	fbCoeRead(bExecute:= FALSE);
		IF NOT fbCoeRead.bBusy THEN					(* Baustein ist durchgelaufen *)
		IF fbCoeRead.bError THEN				(* Wenn ein Error vorliegt, wird dieser ausgegeben *)
			nLastErrIDTemp 
				:= fbCoeRead.nErrID;
			bCoeReadError := TRUE;
		ELSE
			IF nReadBuf.0 THEN
				arrSafetyKlemmeInfo[nAktKlemme].arrFehler[nFehlerIdx] := TRUE;
				arrSafetyKlemmeInfo[nAktKlemme].arrFehlertext[nFehlerIdx] := 
					CONCAT('Temperaturfehler der Safety-Klemme! Uebertemperatur µC1! Adresse: ',
						arrSafetyKlemmeInfo[nAktKlemme].sName);
				nFehlerIdx := nFehlerIdx + 1;
			END_IF	
			IF nReadBuf.1 THEN
				arrSafetyKlemmeInfo[nAktKlemme].arrFehler[nFehlerIdx] := TRUE;
				arrSafetyKlemmeInfo[nAktKlemme].arrFehlertext[nFehlerIdx] := 
					CONCAT('Temperaturfehler der Safety-Klemme! Uebertemperatur µC2! Adresse: ',
						arrSafetyKlemmeInfo[nAktKlemme].sName);
				nFehlerIdx := nFehlerIdx + 1;	
			END_IF	
			IF  nReadBuf.2 THEN
				arrSafetyKlemmeInfo[nAktKlemme].arrFehler[nFehlerIdx] := TRUE;
				arrSafetyKlemmeInfo[nAktKlemme].arrFehlertext[nFehlerIdx] := 
					CONCAT('Temperaturfehler der Safety-Klemme! Uebertemperatur der Ausgangsplatine! Adresse: ',
						arrSafetyKlemmeInfo[nAktKlemme].sName);
				nFehlerIdx := nFehlerIdx + 1;	
			END_IF	
			IF nReadBuf.3 THEN
				arrSafetyKlemmeInfo[nAktKlemme].arrFehler[nFehlerIdx] := TRUE;
				arrSafetyKlemmeInfo[nAktKlemme].arrFehlertext[nFehlerIdx] := 
					CONCAT('Temperaturfehler der Safety-Klemme! Untertemperatur µC1! Adresse: ',
						arrSafetyKlemmeInfo[nAktKlemme].sName);
				nFehlerIdx := nFehlerIdx + 1;	
			END_IF
			(*Fehler am Ausgang - Open Load oder Mindeststrom unterschritten / Höchststrom überschritten*)
			IF nReadBuf.4 THEN
				arrSafetyKlemmeInfo[nAktKlemme].arrFehler[nFehlerIdx] := TRUE;
				arrSafetyKlemmeInfo[nAktKlemme].arrFehlertext[nFehlerIdx] := 
					CONCAT('Temperaturfehler der Safety-Klemme! Untertemperatur µC1! Adresse: ',
						arrSafetyKlemmeInfo[nAktKlemme].sName);
				nFehlerIdx := nFehlerIdx + 1;	
			END_IF
			IF nReadBuf.5 THEN
				arrSafetyKlemmeInfo[nAktKlemme].arrFehler[nFehlerIdx] := TRUE;
				arrSafetyKlemmeInfo[nAktKlemme].arrFehlertext[nFehlerIdx] := 
					CONCAT('Temperaturfehler der Safety-Klemme! Untertemperatur der Ausgangsplatine! Adresse: ',
						arrSafetyKlemmeInfo[nAktKlemme].sName);
				nFehlerIdx := nFehlerIdx + 1;	
			END_IF	
			IF nReadBuf.6 THEN
				arrSafetyKlemmeInfo[nAktKlemme].arrFehler[nFehlerIdx] := TRUE;
				arrSafetyKlemmeInfo[nAktKlemme].arrFehlertext[nFehlerIdx] := 
					CONCAT('Temperaturfehler der Safety-Klemme! Temperaturdifferenz auf der Prozessorplatine ist zu groß! Adresse: ',
						arrSafetyKlemmeInfo[nAktKlemme].sName);
				nFehlerIdx := nFehlerIdx + 1;	
			END_IF	
			IF nReadBuf.7 THEN
				arrSafetyKlemmeInfo[nAktKlemme].arrFehler[nFehlerIdx] := TRUE;
				arrSafetyKlemmeInfo[nAktKlemme].arrFehlertext[nFehlerIdx] := 
					CONCAT('Temperaturfehler der Safety-Klemme! Temperaturdifferenz zwischen den Platinen ist zu groß! Adresse: ',
						arrSafetyKlemmeInfo[nAktKlemme].sName);
				nFehlerIdx := nFehlerIdx + 1;	
			END_IF	
			bCoeReadError := FALSE;
		END_IF
		nStateDatenAuslesen := 0;	
		arrSafetyKlemmeInfo[nAktKlemme].nAnzFehler := nFehlerIdx;
		nFehlerIdx := 0;
		bBusy := FALSE;	
	END_IF
END_CASE

sKlarTextCoeMeldung	:= F_AdsErrorIdToString(I_nErrorID:=nLastErrIDTemp);
END_ACTION

ACTION e_EL2911:

// 16#10F3 ist der Index für den Diag-History-Reiter in der online-Ansicht im EA-Baum
// 16#01: Subindex für das Maximum an Meldungen
// 16#02: Subindex für die neuste Meldung
// 16#03: Subindex für die neuste quittierte Meldung
// 16#04: Subindex eine neue Meldung vorhanden
// 16#05: Subindex für allgemeine Flags
// 16#06 - 16#45: Subindexe für die Meldungen

// Weitere Diagnoseobjekte:
// 16#F984 ist der Index für Device System Data vom Controller 1
// 16#02: Subindex für die Temperatur
// 16#F985 ist der Index für Device System Data vom Controller 2
// 16#02: Subindex für die Temperatur
// Sollten aber auch alle in der Diag History stehen.

// ModuleFault:
// 16#6002:01 Ch1
// 16#6012:01 Ch2
// 16#6022:01 Ch3
// 16#6032:01 Ch4
// 16#6042:01 Ch5
// 16#6052:01 Ch6
// 16#6062:01 Ch7
// 16#6072:01 Ch8

// Eine richtige Diagnose der TwinSAFE-Ein-/ und Ausgänge ist nicht mehr über die CoE-Objekte möglich. Das muss über die DiagHistory gemacht werden. GGf. ist das bald in der HMI
CASE nStateDatenAuslesen OF
	
0:	// EL2912 Diagnose init 
	bBusy 			:= TRUE;	// Solange diese Bit an ist, wird diese Aktion aufgerufen
	nChannelDiag	:= 1;	// Immer bei Kanal 1 beginnen.
	MEMSET(ADR(arrModuleFault),0,SIZEOF(arrModuleFault));	// Rücksetzen
	MEMSET(ADR(arrModuleFaultLink),0,SIZEOF(arrModuleFaultLink));	// Rücksetzen
	
	nStateDatenAuslesen	:= nStateDatenAuslesen +1;
	
1:	// Module Fault der einzelnen Kanäle auslesen: Index errechnen
	
	nCoeIndex		:= 16#6002 + ((nChannelDiag-1)* 16#10);	// Index für ModuleFault pro Kanal
	nCoESubIndex	:= 16#01;	// Index der neusten Meldung
	nStateDatenAuslesen	:= nStateDatenAuslesen +1;
	
2:	// Module Fault der einzelnen Kanäle auslesen: Lesen starten

	fbCoeRead(
		sNetId		:= sEtherCatNetID,
		nSlaveAddr 	:= arrSafetyKlemmeInfo[nAktKlemme].nAdresse,
		nIndex		:= nCoEIndex,
		nSubIndex 	:= nCoESubIndex,
		pDstBuf		:= ADR(nDiagMessage),
		cbBufLen		:= SIZEOF(nDiagMessage),
		bExecute		:= TRUE,

		bError		=> bCoeReadError,
		nErrId		=> nCoeReadErrId
	);
	nStateDatenAuslesen := nStateDatenAuslesen + 1;

3:	// Module Fault der einzelnen Kanäle auslesen: Warten auf gelesen

	fbCoeRead(bExecute:= FALSE);

	IF NOT fbCoeRead.bBusy
	THEN	// Baustein ist durchgelaufen
		IF fbCoeRead.bError
		THEN	// Wenn ein Error vorliegt, wird dieser ausgegeben
			nLastErrIDTemp := fbCoeRead.nErrID;	// Error-ID des CoE Reads wird gespeichert
			bCoeReadError := TRUE;
		ELSE
			bCoeReadError := FALSE;
		END_IF
		
		nStateDatenAuslesen := nStateDatenAuslesen + 1;
	END_IF
	
4:	// Module Fault der einzelnen Kanäle auslesen: Lesen auswerten

	arrModuleFault[nChannelDiag]	:= nDiagMessage <> 0;
	
	IF nChannelDiag = 1
	THEN
		nStateDatenAuslesen := 11;
		nChannelDiag	:= 1;
	ELSE
		nChannelDiag	:= nChannelDiag +1;
		nStateDatenAuslesen := 1;
	END_IF

11:	// Module Fault Link der einzelnen Kanäle auslesen: Index errechnen

// ModuleFaultLink:
// 16#8000:07 Ch1
// 16#8010:07 Ch2
// 16#8020:07 Ch3
// 16#8030:07 Ch4
// 16#8040:07 Ch5
// 16#8050:07 Ch6
// 16#8060:07 Ch7
// 16#8070:07 Ch8

	nCoeIndex		:= 16#8000 + ((nChannelDiag-1)* 16#10);	// Index für ModuleFaultLink pro Kanal
	nCoESubIndex	:= 16#07;
	nStateDatenAuslesen	:= nStateDatenAuslesen +1;
	
12:	// Module Fault Link der einzelnen Kanäle auslesen: Lesen starten

	fbCoeRead(
		sNetId		:= sEtherCatNetID,
		nSlaveAddr 	:= arrSafetyKlemmeInfo[nAktKlemme].nAdresse,
		nIndex		:= nCoEIndex,
		nSubIndex 	:= nCoESubIndex,
		pDstBuf		:= ADR(nDiagMessage),
		cbBufLen		:= SIZEOF(nDiagMessage),
		bExecute		:= TRUE,

		bError		=> bCoeReadError,
		nErrId		=> nCoeReadErrId
	);
	nStateDatenAuslesen := nStateDatenAuslesen + 1;

13:	// Module Fault Link der einzelnen Kanäle auslesen: Warten auf gelesen

	fbCoeRead(bExecute:= FALSE);

	IF NOT fbCoeRead.bBusy
	THEN	// Baustein ist durchgelaufen
		IF fbCoeRead.bError
		THEN	// Wenn ein Error vorliegt, wird dieser ausgegeben
			nLastErrIDTemp := fbCoeRead.nErrID;	// Error-ID des CoE Reads wird gespeichert
			bCoeReadError := TRUE;
		ELSE
			bCoeReadError := FALSE;
		END_IF
		
		nStateDatenAuslesen := nStateDatenAuslesen + 1;
	END_IF
	
14:	// Module Fault Link der einzelnen Kanäle auslesen: Lesen auswerten

	arrModuleFaultLink[nChannelDiag]	:= nDiagMessage <> 0;
	
	IF nChannelDiag = 1
	THEN
		nStateDatenAuslesen := 21;
		nChannelDiag	:= 1;
	ELSE
		nChannelDiag	:= nChannelDiag +1;
		nStateDatenAuslesen := 11;
	END_IF
	
21:	// ModuleFault gesammelt auswerten.

	bModuleFaultActive	:= FALSE;
	FOR nChannelDiag := 1 TO 1 DO
		IF arrModuleFault[nChannelDiag]
		THEN
			bModuleFaultActive	:= TRUE;
		END_IF
	END_FOR
	
	nStateDatenAuslesen := nStateDatenAuslesen + 1;
	
22:	// Fehlermeldung auswerten

	FOR nChannelDiag := 1 TO 1 DO
		IF arrModuleFault[nChannelDiag]
			AND arrModuleFaultLink[nChannelDiag]
		THEN	// Modulfehler mit aktivem ModuleFaultLink
		
			arrSafetyKlemmeInfo[nAktKlemme].arrFehler[nFehlerIdx] := TRUE;
			arrSafetyKlemmeInfo[nAktKlemme].arrFehlertext[nFehlerIdx] := 
				CONCAT('ModuleFault bei Klemme: ',
				CONCAT(arrSafetyKlemmeInfo[nAktKlemme].sName,
				CONCAT(' Kanal: ',
				CONCAT(TO_STRING(nChannelDiag),' Bei aktivem ModuleFaultLink. Der Fehler kann aber auch an einem anderen Kanal liegen.'))));
			nFehlerIdx := nFehlerIdx + 1;
		ELSIF arrModuleFault[nChannelDiag]
		THEN	// Modulfehler ohne ModuleFaultLink. Das heißt, dass der Fehler definitiv an diesem Kanal liegt.
		
			arrSafetyKlemmeInfo[nAktKlemme].arrFehler[nFehlerIdx] := TRUE;
			arrSafetyKlemmeInfo[nAktKlemme].arrFehlertext[nFehlerIdx] := 
				CONCAT('ModuleFault bei Klemme: ',
				CONCAT(arrSafetyKlemmeInfo[nAktKlemme].sName,
				CONCAT(' Kanal: ',TO_STRING(nChannelDiag))));
			nFehlerIdx := nFehlerIdx + 1;
		END_IF
	END_FOR
	
	nStateDatenAuslesen := 99;	// Fertig
	
99:	// Fertig mit auslesen
	
	arrSafetyKlemmeInfo[nAktKlemme].nAnzFehler := nFehlerIdx;
	nStateDatenAuslesen := 0;
	nFehlerIdx := 0; 
	bBusy := FALSE;

END_CASE
END_ACTION

ACTION e_EL2912:

// 16#10F3 ist der Index für den Diag-History-Reiter in der online-Ansicht im EA-Baum
// 16#01: Subindex für das Maximum an Meldungen
// 16#02: Subindex für die neuste Meldung
// 16#03: Subindex für die neuste quittierte Meldung
// 16#04: Subindex eine neue Meldung vorhanden
// 16#05: Subindex für allgemeine Flags
// 16#06 - 16#45: Subindexe für die Meldungen

// Weitere Diagnoseobjekte:
// 16#F984 ist der Index für Device System Data vom Controller 1
// 16#02: Subindex für die Temperatur
// 16#F985 ist der Index für Device System Data vom Controller 2
// 16#02: Subindex für die Temperatur
// Sollten aber auch alle in der Diag History stehen.

// ModuleFault:
// 16#6002:01 Ch1
// 16#6012:01 Ch2
// 16#6022:01 Ch3
// 16#6032:01 Ch4
// 16#6042:01 Ch5
// 16#6052:01 Ch6
// 16#6062:01 Ch7
// 16#6072:01 Ch8

// Eine richtige Diagnose der TwinSAFE-Ein-/ und Ausgänge ist nicht mehr über die CoE-Objekte möglich. Das muss über die DiagHistory gemacht werden. GGf. ist das bald in der HMI
CASE nStateDatenAuslesen OF
	
0:	// EL2912 Diagnose init 
	bBusy 			:= TRUE;	// Solange diese Bit an ist, wird diese Aktion aufgerufen
	nChannelDiag	:= 1;	// Immer bei Kanal 1 beginnen.
	MEMSET(ADR(arrModuleFault),0,SIZEOF(arrModuleFault));	// Rücksetzen
	MEMSET(ADR(arrModuleFaultLink),0,SIZEOF(arrModuleFaultLink));	// Rücksetzen
	
	nStateDatenAuslesen	:= nStateDatenAuslesen +1;
	
1:	// Module Fault der einzelnen Kanäle auslesen: Index errechnen
	
	nCoeIndex		:= 16#6002 + ((nChannelDiag-1)* 16#10);	// Index für ModuleFault pro Kanal
	nCoESubIndex	:= 16#01;	// Index der neusten Meldung
	nStateDatenAuslesen	:= nStateDatenAuslesen +1;
	
2:	// Module Fault der einzelnen Kanäle auslesen: Lesen starten

	fbCoeRead(
		sNetId		:= sEtherCatNetID,
		nSlaveAddr 	:= arrSafetyKlemmeInfo[nAktKlemme].nAdresse,
		nIndex		:= nCoEIndex,
		nSubIndex 	:= nCoESubIndex,
		pDstBuf		:= ADR(nDiagMessage),
		cbBufLen		:= SIZEOF(nDiagMessage),
		bExecute		:= TRUE,

		bError		=> bCoeReadError,
		nErrId		=> nCoeReadErrId
	);
	nStateDatenAuslesen := nStateDatenAuslesen + 1;

3:	// Module Fault der einzelnen Kanäle auslesen: Warten auf gelesen

	fbCoeRead(bExecute:= FALSE);

	IF NOT fbCoeRead.bBusy
	THEN	// Baustein ist durchgelaufen
		IF fbCoeRead.bError
		THEN	// Wenn ein Error vorliegt, wird dieser ausgegeben
			nLastErrIDTemp := fbCoeRead.nErrID;	// Error-ID des CoE Reads wird gespeichert
			bCoeReadError := TRUE;
		ELSE
			bCoeReadError := FALSE;
		END_IF
		
		nStateDatenAuslesen := nStateDatenAuslesen + 1;
	END_IF
	
4:	// Module Fault der einzelnen Kanäle auslesen: Lesen auswerten

	arrModuleFault[nChannelDiag]	:= nDiagMessage <> 0;
	
	IF nChannelDiag = 2
	THEN
		nStateDatenAuslesen := 11;
		nChannelDiag	:= 1;
	ELSE
		nChannelDiag	:= nChannelDiag +1;
		nStateDatenAuslesen := 1;
	END_IF

11:	// Module Fault Link der einzelnen Kanäle auslesen: Index errechnen

// ModuleFaultLink:
// 16#8000:07 Ch1
// 16#8010:07 Ch2
// 16#8020:07 Ch3
// 16#8030:07 Ch4
// 16#8040:07 Ch5
// 16#8050:07 Ch6
// 16#8060:07 Ch7
// 16#8070:07 Ch8

	nCoeIndex		:= 16#8000 + ((nChannelDiag-1)* 16#10);	// Index für ModuleFaultLink pro Kanal
	nCoESubIndex	:= 16#07;
	nStateDatenAuslesen	:= nStateDatenAuslesen +1;
	
12:	// Module Fault Link der einzelnen Kanäle auslesen: Lesen starten

	fbCoeRead(
		sNetId		:= sEtherCatNetID,
		nSlaveAddr 	:= arrSafetyKlemmeInfo[nAktKlemme].nAdresse,
		nIndex		:= nCoEIndex,
		nSubIndex 	:= nCoESubIndex,
		pDstBuf		:= ADR(nDiagMessage),
		cbBufLen		:= SIZEOF(nDiagMessage),
		bExecute		:= TRUE,

		bError		=> bCoeReadError,
		nErrId		=> nCoeReadErrId
	);
	nStateDatenAuslesen := nStateDatenAuslesen + 1;

13:	// Module Fault Link der einzelnen Kanäle auslesen: Warten auf gelesen

	fbCoeRead(bExecute:= FALSE);

	IF NOT fbCoeRead.bBusy
	THEN	// Baustein ist durchgelaufen
		IF fbCoeRead.bError
		THEN	// Wenn ein Error vorliegt, wird dieser ausgegeben
			nLastErrIDTemp := fbCoeRead.nErrID;	// Error-ID des CoE Reads wird gespeichert
			bCoeReadError := TRUE;
		ELSE
			bCoeReadError := FALSE;
		END_IF
		
		nStateDatenAuslesen := nStateDatenAuslesen + 1;
	END_IF
	
14:	// Module Fault Link der einzelnen Kanäle auslesen: Lesen auswerten

	arrModuleFaultLink[nChannelDiag]	:= nDiagMessage <> 0;
	
	IF nChannelDiag = 2
	THEN
		nStateDatenAuslesen := 21;
		nChannelDiag	:= 1;
	ELSE
		nChannelDiag	:= nChannelDiag +1;
		nStateDatenAuslesen := 11;
	END_IF
	
21:	// ModuleFault gesammelt auswerten.

	bModuleFaultActive	:= FALSE;
	FOR nChannelDiag := 1 TO 2 DO
		IF arrModuleFault[nChannelDiag]
		THEN
			bModuleFaultActive	:= TRUE;
		END_IF
	END_FOR
	
	nStateDatenAuslesen := nStateDatenAuslesen + 1;
	
22:	// Fehlermeldung auswerten

	FOR nChannelDiag := 1 TO 2 DO
		IF arrModuleFault[nChannelDiag]
			AND arrModuleFaultLink[nChannelDiag]
		THEN	// Modulfehler mit aktivem ModuleFaultLink
		
			arrSafetyKlemmeInfo[nAktKlemme].arrFehler[nFehlerIdx] := TRUE;
			arrSafetyKlemmeInfo[nAktKlemme].arrFehlertext[nFehlerIdx] := 
				CONCAT('ModuleFault bei Klemme: ',
				CONCAT(arrSafetyKlemmeInfo[nAktKlemme].sName,
				CONCAT(' Kanal: ',
				CONCAT(TO_STRING(nChannelDiag),' Bei aktivem ModuleFaultLink. Der Fehler kann aber auch an einem anderen Kanal liegen.'))));
			nFehlerIdx := nFehlerIdx + 1;
		ELSIF arrModuleFault[nChannelDiag]
		THEN	// Modulfehler ohne ModuleFaultLink. Das heißt, dass der Fehler definitiv an diesem Kanal liegt.
		
			arrSafetyKlemmeInfo[nAktKlemme].arrFehler[nFehlerIdx] := TRUE;
			arrSafetyKlemmeInfo[nAktKlemme].arrFehlertext[nFehlerIdx] := 
				CONCAT('ModuleFault bei Klemme: ',
				CONCAT(arrSafetyKlemmeInfo[nAktKlemme].sName,
				CONCAT(' Kanal: ',TO_STRING(nChannelDiag))));
			nFehlerIdx := nFehlerIdx + 1;
		END_IF
	END_FOR
	
	nStateDatenAuslesen := 99;	// Fertig
	
99:	// Fertig mit auslesen
	
	arrSafetyKlemmeInfo[nAktKlemme].nAnzFehler := nFehlerIdx;
	nStateDatenAuslesen := 0;
	nFehlerIdx := 0; 
	bBusy := FALSE;

END_CASE
END_ACTION

ACTION e_EP2918:

// 16#10F3 ist der Index für den Diag-History-Reiter in der online-Ansicht im EA-Baum
// 16#01: Subindex für das Maximum an Meldungen
// 16#02: Subindex für die neuste Meldung
// 16#03: Subindex für die neuste quittierte Meldung
// 16#04: Subindex eine neue Meldung vorhanden
// 16#05: Subindex für allgemeine Flags
// 16#06 - 16#45: Subindexe für die Meldungen

// Weitere Diagnoseobjekte:
// 16#F984 ist der Index für Device System Data vom Controller 1
// 16#02: Subindex für die Temperatur
// 16#F985 ist der Index für Device System Data vom Controller 2
// 16#02: Subindex für die Temperatur
// Sollten aber auch alle in der Diag History stehen.

// ModuleFault:
// 16#6002:01 Ch1
// 16#6012:01 Ch2
// 16#6022:01 Ch3
// 16#6032:01 Ch4
// 16#6042:01 Ch5
// 16#6052:01 Ch6
// 16#6062:01 Ch7
// 16#6072:01 Ch8

// Eine richtige Diagnose der TwinSAFE-Ein-/ und Ausgänge ist nicht mehr über die CoE-Objekte möglich. Das muss über die DiagHistory gemacht werden. GGf. ist das bald in der HMI
CASE nStateDatenAuslesen OF
	
0:	// EL2912 Diagnose init 
	bBusy 			:= TRUE;	// Solange diese Bit an ist, wird diese Aktion aufgerufen
	nChannelDiag	:= 1;	// Immer bei Kanal 1 beginnen.
	MEMSET(ADR(arrModuleFault),0,SIZEOF(arrModuleFault));	// Rücksetzen
	MEMSET(ADR(arrModuleFaultLink),0,SIZEOF(arrModuleFaultLink));	// Rücksetzen
	
	nStateDatenAuslesen	:= nStateDatenAuslesen +1;
	
1:	// Module Fault der einzelnen Kanäle auslesen: Index errechnen
	
	nCoeIndex		:= 16#6002 + ((nChannelDiag-1)* 16#10);	// Index für ModuleFault pro Kanal
	nCoESubIndex	:= 16#01;	// Index der neusten Meldung
	nStateDatenAuslesen	:= nStateDatenAuslesen +1;
	
2:	// Module Fault der einzelnen Kanäle auslesen: Lesen starten

	fbCoeRead(
		sNetId		:= sEtherCatNetID,
		nSlaveAddr 	:= arrSafetyKlemmeInfo[nAktKlemme].nAdresse,
		nIndex		:= nCoEIndex,
		nSubIndex 	:= nCoESubIndex,
		pDstBuf		:= ADR(nDiagMessage),
		cbBufLen		:= SIZEOF(nDiagMessage),
		bExecute		:= TRUE,

		bError		=> bCoeReadError,
		nErrId		=> nCoeReadErrId
	);
	nStateDatenAuslesen := nStateDatenAuslesen + 1;

3:	// Module Fault der einzelnen Kanäle auslesen: Warten auf gelesen

	fbCoeRead(bExecute:= FALSE);

	IF NOT fbCoeRead.bBusy
	THEN	// Baustein ist durchgelaufen
		IF fbCoeRead.bError
		THEN	// Wenn ein Error vorliegt, wird dieser ausgegeben
			nLastErrIDTemp := fbCoeRead.nErrID;	// Error-ID des CoE Reads wird gespeichert
			bCoeReadError := TRUE;
		ELSE
			bCoeReadError := FALSE;
		END_IF
		
		nStateDatenAuslesen := nStateDatenAuslesen + 1;
	END_IF
	
4:	// Module Fault der einzelnen Kanäle auslesen: Lesen auswerten

	arrModuleFault[nChannelDiag]	:= nDiagMessage <> 0;
	
	IF nChannelDiag = 8
	THEN
		nStateDatenAuslesen := 11;
		nChannelDiag	:= 1;
	ELSE
		nChannelDiag	:= nChannelDiag +1;
		nStateDatenAuslesen := 1;
	END_IF

11:	// Module Fault Link der einzelnen Kanäle auslesen: Index errechnen

// ModuleFaultLink:
// 16#8000:07 Ch1
// 16#8010:07 Ch2
// 16#8020:07 Ch3
// 16#8030:07 Ch4
// 16#8040:07 Ch5
// 16#8050:07 Ch6
// 16#8060:07 Ch7
// 16#8070:07 Ch8

	nCoeIndex		:= 16#8000 + ((nChannelDiag-1)* 16#10);	// Index für ModuleFaultLink pro Kanal
	nCoESubIndex	:= 16#07;
	nStateDatenAuslesen	:= nStateDatenAuslesen +1;
	
12:	// Module Fault Link der einzelnen Kanäle auslesen: Lesen starten

	fbCoeRead(
		sNetId		:= sEtherCatNetID,
		nSlaveAddr 	:= arrSafetyKlemmeInfo[nAktKlemme].nAdresse,
		nIndex		:= nCoEIndex,
		nSubIndex 	:= nCoESubIndex,
		pDstBuf		:= ADR(nDiagMessage),
		cbBufLen		:= SIZEOF(nDiagMessage),
		bExecute		:= TRUE,

		bError		=> bCoeReadError,
		nErrId		=> nCoeReadErrId
	);
	nStateDatenAuslesen := nStateDatenAuslesen + 1;

13:	// Module Fault Link der einzelnen Kanäle auslesen: Warten auf gelesen

	fbCoeRead(bExecute:= FALSE);

	IF NOT fbCoeRead.bBusy
	THEN	// Baustein ist durchgelaufen
		IF fbCoeRead.bError
		THEN	// Wenn ein Error vorliegt, wird dieser ausgegeben
			nLastErrIDTemp := fbCoeRead.nErrID;	// Error-ID des CoE Reads wird gespeichert
			bCoeReadError := TRUE;
		ELSE
			bCoeReadError := FALSE;
		END_IF
		
		nStateDatenAuslesen := nStateDatenAuslesen + 1;
	END_IF
	
14:	// Module Fault Link der einzelnen Kanäle auslesen: Lesen auswerten

	arrModuleFaultLink[nChannelDiag]	:= nDiagMessage <> 0;
	
	IF nChannelDiag = 8
	THEN
		nStateDatenAuslesen := 21;
		nChannelDiag	:= 1;
	ELSE
		nChannelDiag	:= nChannelDiag +1;
		nStateDatenAuslesen := 11;
	END_IF
	
21:	// ModuleFault gesammelt auswerten.

	bModuleFaultActive	:= FALSE;
	FOR nChannelDiag := 1 TO 8 DO
		IF arrModuleFault[nChannelDiag]
		THEN
			bModuleFaultActive	:= TRUE;
		END_IF
	END_FOR
	
	nStateDatenAuslesen := nStateDatenAuslesen + 1;
	
22:	// Fehlermeldung auswerten

	FOR nChannelDiag := 1 TO 8 DO
		IF arrModuleFault[nChannelDiag]
			AND arrModuleFaultLink[nChannelDiag]
		THEN	// Modulfehler mit aktivem ModuleFaultLink
		
			arrSafetyKlemmeInfo[nAktKlemme].arrFehler[nFehlerIdx] := TRUE;
			arrSafetyKlemmeInfo[nAktKlemme].arrFehlertext[nFehlerIdx] := 
				CONCAT('ModuleFault bei Klemme: ',
				CONCAT(arrSafetyKlemmeInfo[nAktKlemme].sName,
				CONCAT(' Kanal: ',
				CONCAT(TO_STRING(nChannelDiag),' Bei aktivem ModuleFaultLink. Der Fehler kann aber auch an einem anderen Kanal liegen.'))));
			nFehlerIdx := nFehlerIdx + 1;
		ELSIF arrModuleFault[nChannelDiag]
		THEN	// Modulfehler ohne ModuleFaultLink. Das heißt, dass der Fehler definitiv an diesem Kanal liegt.
		
			arrSafetyKlemmeInfo[nAktKlemme].arrFehler[nFehlerIdx] := TRUE;
			arrSafetyKlemmeInfo[nAktKlemme].arrFehlertext[nFehlerIdx] := 
				CONCAT('ModuleFault bei Klemme: ',
				CONCAT(arrSafetyKlemmeInfo[nAktKlemme].sName,
				CONCAT(' Kanal: ',TO_STRING(nChannelDiag))));
			nFehlerIdx := nFehlerIdx + 1;
		END_IF
	END_FOR
	
	nStateDatenAuslesen := 99;	// Fertig
	
99:	// Fertig mit auslesen
	
	arrSafetyKlemmeInfo[nAktKlemme].nAnzFehler := nFehlerIdx;
	nStateDatenAuslesen := 0;
	nFehlerIdx := 0; 
	bBusy := FALSE;

END_CASE
END_ACTION

ACTION f_AX5805:
CASE nStateDatenAuslesen OF
0:
	(*Auslesen der Anzahl der Achsen*)
	bBusy				:= TRUE;	
	nCoeIndex		:= 16#2F00; (*Anzahl der Achsen*)
	nCoESubIndex	:= 16#1;
	
	fbCoeRead(
	sNetId		:= sEtherCatNetID,
	nSlaveAddr 	:= arrSafetyKlemmeInfo[nAktKlemme].nAdresse,
	nIndex		:= nCoEIndex,
	nSubIndex 	:= nCoESubIndex,
	pDstBuf		:= ADR(nReadBuf),
	cbBufLen		:= SIZEOF(nReadBuf),
	bExecute		:= TRUE,

	bError		=> bCoeReadError,
	nErrId		=> nCoeReadErrId
	);
	
	fbCoeRead(bExecute:= FALSE);
	nAnzahlAchsen := UDINT_TO_INT(nReadBuf);
	
	IF NOT fbCoeRead.bBusy THEN
		nStateDatenAuslesen := nStateDatenAuslesen + 1;
	END_IF

1:	
	IF nAktAChse < nAnzahlAchsen THEN
		IF nAktAchse = 0 THEN
			  nAktAchse := 1;
	   END_IF
		
		nCoeIndex		:= 16#FA10; (*Grund der Abschaltung*)
		IF nAktAchse = 1 THEN 
			nCoESubIndex := 16#07;	(*Index Achse 1*)
		ELSE
			nCoeSubIndex := 16#08;	(*Index Achse 2*)
		END_IF
		 
		 fbCoeRead(
		 sNetId		:= sEtherCatNetID,
		 nSlaveAddr := arrSafetyKlemmeInfo[nAktKlemme].nAdresse,
		 nIndex		:= nCoEIndex,
		 nSubIndex 	:= nCoESubIndex,
		 pDstBuf		:= ADR(nReadBuf),
		 cbBufLen		:= SIZEOF(nReadBuf),
		 bExecute		:= TRUE,
	 
		 bError		=> bCoeReadError,
		 nErrId		=> nCoeReadErrId
		 );
			 
		 fbCoeRead(bExecute:= FALSE);
	 
		 IF NOT fbCoeRead.bBusy THEN				(* Baustein ist durchgelaufen *)
			 IF fbCoeRead.bError THEN				(* Wenn ein Error vorliegt, wird dieser ausgegeben; 0 = kein Fehler, 1= Eingang 1; 2= Eingang 2; 3= Eingang 3; 4 = Eingang 4*)
				 nLastErrIDTemp 
					 := fbCoeRead.nErrID;
				 bCoeReadError := TRUE;
			 ELSE
		 (*Fehler-Meldungen - Grund der Abschaltung CoE Objekt 0xFA10:07 und 0xFA10:08*)
		 (*Fehlermeldung aus AX5805.pdf Stand 03.12.2013 - S.101*)
			IF nReadBuf >= 16#100
			 AND nReadBuf < 16#200 THEN
				arrSafetyKlemmeInfo[nAktKlemme].arrFehler[nFehlerIdx] := TRUE;
				arrSafetyKlemmeInfo[nAktKlemme].arrFehlertext[nFehlerIdx] := 
					 CONCAT('AX5805: Das Statuswort wurde falsch berechnet! Achse: ',
					 CONCAT(INT_TO_STRING(nAktAchse),
					 CONCAT('Adresse: ',
						arrSafetyKlemmeInfo[nAktKlemme].sName)));
				nFehlerIdx := nFehlerIdx + 1;
			ELSIF nReadBuf >= 16#200
			 AND nReadBuf < 16#300 THEN
				arrSafetyKlemmeInfo[nAktKlemme].arrFehler[nFehlerIdx] := TRUE;
				arrSafetyKlemmeInfo[nAktKlemme].arrFehlertext[nFehlerIdx] := 
					 CONCAT('AX5805: Die Parameter sind fehlerhaft, wurden noch nicht geladen oder der AX5805 wurde noch nicht zurueckgesetzt (Error_Ack)! Achse: ',
					 CONCAT(INT_TO_STRING(nAktAchse),
					 CONCAT('Adresse: ',
						arrSafetyKlemmeInfo[nAktKlemme].sName)));
				nFehlerIdx := nFehlerIdx + 1;	
			ELSIF nReadBuf >= 16#300
			 AND nReadBuf < 16#400 THEN
				arrSafetyKlemmeInfo[nAktKlemme].arrFehler[nFehlerIdx] := TRUE;
				arrSafetyKlemmeInfo[nAktKlemme].arrFehlertext[nFehlerIdx] := 
					 CONCAT('AX5805: FSOE-Protokoll nicht im State DATA! Achse: ',
					 CONCAT(INT_TO_STRING(nAktAchse),
					 CONCAT('Adresse: ',
						arrSafetyKlemmeInfo[nAktKlemme].sName)));
				nFehlerIdx := nFehlerIdx + 1;
			ELSIF nReadBuf >= 16#400
			 AND nReadBuf < 16#500 THEN
				arrSafetyKlemmeInfo[nAktKlemme].arrFehler[nFehlerIdx] := TRUE;
				arrSafetyKlemmeInfo[nAktKlemme].arrFehlertext[nFehlerIdx] := 
					 CONCAT('AX5805: FSOE-Protokoll nicht im State DATA! Achse: ',
					 CONCAT(INT_TO_STRING(nAktAchse),
					 CONCAT('Adresse: ',
						arrSafetyKlemmeInfo[nAktKlemme].sName)));
				nFehlerIdx := nFehlerIdx + 1;
			 ELSIF nReadBuf >= 16#500
				 AND nReadBuf < 16#600 THEN
					 arrSafetyKlemmeInfo[nAktKlemme].arrFehler[nFehlerIdx] := TRUE;
					 arrSafetyKlemmeInfo[nAktKlemme].arrFehlertext[nFehlerIdx] := 
						  CONCAT('AX5805: FSOE-Protokoll nicht im State DATA! Achse: ',
						  CONCAT(INT_TO_STRING(nAktAchse),
						  CONCAT('Adresse: ',
							 arrSafetyKlemmeInfo[nAktKlemme].sName)));	
					 nFehlerIdx := nFehlerIdx + 1;
			 ELSIF nReadBuf >= 16#600
				 AND nReadBuf < 16#700 THEN
					 arrSafetyKlemmeInfo[nAktKlemme].arrFehler[nFehlerIdx] := TRUE;
					 arrSafetyKlemmeInfo[nAktKlemme].arrFehlertext[nFehlerIdx] := 
						  CONCAT('AX5805: FSOE-Protokoll nicht im State DATA! Achse: ',
						  CONCAT(INT_TO_STRING(nAktAchse),
						  CONCAT('Adresse: ',
							 arrSafetyKlemmeInfo[nAktKlemme].sName)));	
					 nFehlerIdx := nFehlerIdx + 1;
			 ELSIF nReadBuf >= 16#700
				 AND nReadBuf < 16#800 THEN
					 arrSafetyKlemmeInfo[nAktKlemme].arrFehler[nFehlerIdx] := TRUE;
					 arrSafetyKlemmeInfo[nAktKlemme].arrFehlertext[nFehlerIdx] := 
						  CONCAT('AX5805: FSOE-Protokoll nicht im State DATA! Achse: ',
						  CONCAT(INT_TO_STRING(nAktAchse),
						  CONCAT('Adresse: ',
							 arrSafetyKlemmeInfo[nAktKlemme].sName)));	
					 nFehlerIdx := nFehlerIdx + 1;
			 ELSIF nReadBuf >= 16#800
				 AND nReadBuf < 16#900 THEN
					 arrSafetyKlemmeInfo[nAktKlemme].arrFehler[nFehlerIdx] := TRUE;
					 arrSafetyKlemmeInfo[nAktKlemme].arrFehlertext[nFehlerIdx] := 
						  CONCAT('AX5805: FSOE-Protokoll nicht im State DATA! Achse: ',
						  CONCAT(INT_TO_STRING(nAktAchse),
						  CONCAT('Adresse: ',
							 arrSafetyKlemmeInfo[nAktKlemme].sName)));	
					 nFehlerIdx := nFehlerIdx + 1;
			 ELSIF nReadBuf >= 16#5000
				 AND nReadBuf < 16#6800 THEN
					 arrSafetyKlemmeInfo[nAktKlemme].arrFehler[nFehlerIdx] := TRUE;
					 arrSafetyKlemmeInfo[nAktKlemme].arrFehlertext[nFehlerIdx] := 
						  CONCAT('AX5805: FSOE-Protokoll nicht im State DATA! Achse: ',
						  CONCAT(INT_TO_STRING(nAktAchse),
						  CONCAT('Adresse: ',
							 arrSafetyKlemmeInfo[nAktKlemme].sName)));	
					 nFehlerIdx := nFehlerIdx + 1;
			 ELSIF nReadBuf >= 16#6800
				 AND nReadBuf < 16#8000 THEN
					 arrSafetyKlemmeInfo[nAktKlemme].arrFehler[nFehlerIdx] := TRUE;
					 arrSafetyKlemmeInfo[nAktKlemme].arrFehlertext[nFehlerIdx] := 
						  CONCAT('AX5805: FSOE-Protokoll nicht im State DATA! Achse: ',
						  CONCAT(INT_TO_STRING(nAktAchse),
						  CONCAT('Adresse: ',
							 arrSafetyKlemmeInfo[nAktKlemme].sName)));	
					 nFehlerIdx := nFehlerIdx + 1;
			 ELSIF nReadBuf >= 16#8000
				 AND nReadBuf < 16#9000 THEN
					 arrSafetyKlemmeInfo[nAktKlemme].arrFehler[nFehlerIdx] := TRUE;
					 arrSafetyKlemmeInfo[nAktKlemme].arrFehlertext[nFehlerIdx] := 
						  CONCAT('AX5805: FSOE-Protokoll nicht im State DATA! Achse: ',
						  CONCAT(INT_TO_STRING(nAktAchse),
						  CONCAT('Adresse: ',
							 arrSafetyKlemmeInfo[nAktKlemme].sName)));	
					 nFehlerIdx := nFehlerIdx + 1;
			 ELSIF nReadBuf >= 16#9000
				 AND nReadBuf < 16#A000 THEN
					 arrSafetyKlemmeInfo[nAktKlemme].arrFehler[nFehlerIdx] := TRUE;
					 arrSafetyKlemmeInfo[nAktKlemme].arrFehlertext[nFehlerIdx] := 
						  CONCAT('AX5805: FSOE-Protokoll nicht im State DATA! Achse: ',
						  CONCAT(INT_TO_STRING(nAktAchse),
						  CONCAT('Adresse: ',
							 arrSafetyKlemmeInfo[nAktKlemme].sName)));	
					 nFehlerIdx := nFehlerIdx + 1;
			 ELSIF nReadBuf >= 16#A000
				 AND nReadBuf < 16#A800 THEN
					 arrSafetyKlemmeInfo[nAktKlemme].arrFehler[nFehlerIdx] := TRUE;
					 arrSafetyKlemmeInfo[nAktKlemme].arrFehlertext[nFehlerIdx] := 
						  CONCAT('AX5805: FSOE-Protokoll nicht im State DATA! Achse: ',
						  CONCAT(INT_TO_STRING(nAktAchse),
						  CONCAT('Adresse: ',
							 arrSafetyKlemmeInfo[nAktKlemme].sName)));	
					 nFehlerIdx := nFehlerIdx + 1;
			 ELSIF nReadBuf >= 16#A800
				 AND nReadBuf < 16#B800 THEN
					 arrSafetyKlemmeInfo[nAktKlemme].arrFehler[nFehlerIdx] := TRUE;
					 arrSafetyKlemmeInfo[nAktKlemme].arrFehlertext[nFehlerIdx] := 
						  CONCAT('AX5805: FSOE-Protokoll nicht im State DATA! Achse: ',
						  CONCAT(INT_TO_STRING(nAktAchse),
						  CONCAT('Adresse: ',
							 arrSafetyKlemmeInfo[nAktKlemme].sName)));	
					 nFehlerIdx := nFehlerIdx + 1;
			 ELSIF nReadBuf >= 16#B800
				 AND nReadBuf < 16#C800 THEN
					 arrSafetyKlemmeInfo[nAktKlemme].arrFehler[nFehlerIdx] := TRUE;
					 arrSafetyKlemmeInfo[nAktKlemme].arrFehlertext[nFehlerIdx] := 
						  CONCAT('AX5805: FSOE-Protokoll nicht im State DATA! Achse: ',
						  CONCAT(INT_TO_STRING(nAktAchse),
						  CONCAT('Adresse: ',
							 arrSafetyKlemmeInfo[nAktKlemme].sName)));	
					 nFehlerIdx := nFehlerIdx + 1;
			 ELSIF nReadBuf >= 16#C800
				 AND nReadBuf < 16#D000 THEN
					 arrSafetyKlemmeInfo[nAktKlemme].arrFehler[nFehlerIdx] := TRUE;
					 arrSafetyKlemmeInfo[nAktKlemme].arrFehlertext[nFehlerIdx] := 
						  CONCAT('AX5805: FSOE-Protokoll nicht im State DATA! Achse: ',
						  CONCAT(INT_TO_STRING(nAktAchse),
						  CONCAT('Adresse: ',
							 arrSafetyKlemmeInfo[nAktKlemme].sName)));	
					 nFehlerIdx := nFehlerIdx + 1;
			 ELSIF nReadBuf >= 16#D000
				 AND nReadBuf < 16#D100 THEN
					 arrSafetyKlemmeInfo[nAktKlemme].arrFehler[nFehlerIdx] := TRUE;
					 arrSafetyKlemmeInfo[nAktKlemme].arrFehlertext[nFehlerIdx] := 
						  CONCAT('AX5805: FSOE-Protokoll nicht im State DATA! Achse: ',
						  CONCAT(INT_TO_STRING(nAktAchse),
						  CONCAT('Adresse: ',
							 arrSafetyKlemmeInfo[nAktKlemme].sName)));	
					 nFehlerIdx := nFehlerIdx + 1;
			 ELSIF nReadBuf >= 16#D100 THEN
				 arrSafetyKlemmeInfo[nAktKlemme].arrFehler[nFehlerIdx] := TRUE;
				 arrSafetyKlemmeInfo[nAktKlemme].arrFehlertext[nFehlerIdx] := 
					 CONCAT('AX5805: FSOE-Protokoll nicht im State DATA! Achse: ',
					 CONCAT(INT_TO_STRING(nAktAchse),
					 CONCAT('Adresse: ',
						 arrSafetyKlemmeInfo[nAktKlemme].sName)));	
				 nFehlerIdx := nFehlerIdx + 1;
			 END_IF
			 bCoeReadError := FALSE;
			END_IF
			IF nAktAchse < nAnzahlAchsen THEN
				 nAktAchse := nAktAchse + 1;
			ELSIF nAktAchse = nAnzahlAchsen THEN
				 nAktAchse := 0;
				 nStateDatenAuslesen := nStateDatenAuslesen + 1;
			 END_IF
		  END_IF
		END_IF

3:
	IF nAktAchse > nAnzahlAchsen THEN 
   	IF nAktAchse = 0 THEN	(*Index der Achse wird in die Zahl der Achse umgewandelt*)
			  nAktAchse := 1;
	   END_IF
		
	 (*Sensortest-Fehler-Überprüfung*)
		 nCoeIndex		:= 16#FA82; (*Index fuer die Diagnose*)
		 IF nAktAchse = 1 THEN 
			 nCoESubIndex := 16#03;	(*Index Achse 1*)
		 ELSE
			 nCoeSubIndex := 16#04;	(*Index Achse 2*)
		 END_IF
		 (*Auslesen der Diagnose-Informationen*)
		 fbCoeRead(
		 sNetId		:= sEtherCatNetID,
		 nSlaveAddr := arrSafetyKlemmeInfo[nAktKlemme].nAdresse,
		 nIndex		:= nCoEIndex,
		 nSubIndex 	:= nCoESubIndex,
		 pDstBuf		:= ADR(nReadBuf),
		 cbBufLen	:= SIZEOF(nReadBuf),
		 bExecute	:= TRUE,
	 
		 bError		=> bCoeReadError,
		 nErrId		=> nCoeReadErrId
		 );
	 
		 fbCoeRead(bExecute:= FALSE);
		 IF NOT fbCoeRead.bBusy THEN				(* Baustein ist durchgelaufen *)
			 IF fbCoeRead.bError THEN				(* Wenn ein Error vorliegt, wird dieser ausgegeben; 0 = kein Fehler, 1= Eingang 1; 2= Eingang 2; 3= Eingang 3; 4 = Eingang 4*)
				 nLastErrIDTemp 
					 := fbCoeRead.nErrID;
				 bCoeReadError := TRUE;
			 ELSE
				(*Fehler-Meldungen - Grund der Abschaltung CoE Objekt 0xFA82:03 und 0xFA82:04*)
		 		(*Fehlermeldung aus AX5805.pdf Stand 03.12.2013 - S.101*)
				 CASE nReadBuf OF
					16#0000:
						;
					16#0001:
						sMeldSpeich
							:= ('AX5805: Die maximale Temperatur wurde überschritten (µC1)!');
					16#0002:
						sMeldSpeich
							:= ('AX5805: Die maximale Temperatur wurde überschritten (µC2)!');
					16#0003:
						sMeldSpeich
							:= ('AX5805: Die minimale Temperatur wurde unterschritten (µC1)!');
					16#0004:
						sMeldSpeich
							:= ('AX5805: Die minimale Temperatur wurde unterschritten (µC2)!');
					16#0101:
						sMeldSpeich
							:= ('AX5805: Die maximale Versorgungsspannung wurde überschritten (3,3 V)!');
					16#0102:
						sMeldSpeich
							:= ('AX5805: Die maximale Versorgungsspannung wurde überschritten (3,3 V)!');
					16#0103:
						sMeldSpeich
							:= ('AX5805: Die minimale Versorgungsspannung wurde unterschritten (3,3 V)!');
					16#0104:
						sMeldSpeich
							:= ('AX5805: Die minimale Versorgungsspannung wurde unterschritten (3,3 V)!');
					16#0201:
						sMeldSpeich
							:= ('AX5805: Die MCTests von µC1 wurden nicht vollstandig in der vorgegebenen Zeit durchgeführt!');
					16#0202:
						sMeldSpeich
							:= ('AX5805: Die MCTests von µC2 wurden nicht vollstandig in der vorgegebenen Zeit durchgeführt!');
					16#0203:
						sMeldSpeich
							:= ('AX5805: Der globale Timer wurde nicht rechtzeitig aktualisiert!');
					16#0204:
						sMeldSpeich
							:= ('AX5805: Der globale Timer wurde nicht rechtzeitig aktualisiert!');
					16#020C:
						sMeldSpeich
							:= ('AX5805: Das TwinSAFE Modul wurde nicht innerhalb der Watchdogzeit aufgerufen!');
					16#020D:
						sMeldSpeich
							:= ('AX5805: Das TwinSAFE Modul wurde nicht innerhalb der Watchdogzeit aufgerufen!');
					16#020E:
						sMeldSpeich
							:= ('AX5805: Bei µC1 ist ein Reset im Betrieb des Kontrollers aufgetreten µC2 wurde dabei nicht zuruckgesetzt!');
					16#0300:
						sMeldSpeich
							:= ('AX5805: Fehler im SerComP24C2 Modul ist bei der Datenübertragung aufgetreten!');
					16#0401 .. 16#040B:
						sMeldSpeich
							:= ('AX5805: Fehler im SerComP24C1 Modul ist bei der Datenübertragung aufgetreten!');
					16#0501 .. 16#507:
						sMeldSpeich
							:= ('AX5805: Ein Fehler in der Kommunikation mit einem der Temperatursensoren ist aufgetreten!');
					16#0601:
						sMeldSpeich
							:= ('AX5805: Die von µC1 und µC2 ausgegebenen Werte unterscheiden sich!');
					16#0602:
						sMeldSpeich
							:= ('AX5805: Die von µC1 und µC2 ausgegebenen Werte unterscheiden sich!');
					16#0700:
						sMeldSpeich
							:= ('AX5805: Die minimale FPGA Versorgungsspannung wurde unterschritten (5 V)!');
					16#0701:
						sMeldSpeich
							:= ('AX5805: Die maximale FPGA Versorgungsspannung wurde unterschritten (5 V)!');
					16#0710:
						sMeldSpeich
							:= ('AX5805: Bei den Feedback-Kanalen von µC1 wurde ein Fehler detektiert!');
					16#0711:
						sMeldSpeich
							:= ('AX5805: Bei den Feedback-Kanalen von µC2 wurde ein Fehler detektiert!');
					16#0720:
						sMeldSpeich
							:= ('AX5805: Allgemeiner Parameterfehler µC1!');
					16#0721:
						sMeldSpeich
							:= ('AX5805: Allgemeiner Parameterfehler µC2!');
					16#0722:
						sMeldSpeich
							:= ('AX5805: Parameter: Unbekannter Parameterindex µC1 Drive Profile!');
					16#0723:
						sMeldSpeich
							:= ('AX5805: Parameter: Unbekannter Parameterindex µC1 Hersteller spezifisch!');
					16#0724:
						sMeldSpeich
							:= ('AX5805: Parameter: Unbekannter Parameterindex µC2 Drive Profile!');
					16#0725:
						sMeldSpeich
							:= ('AX5805: Parameter: Unbekannter Parameterindex µC2 Drive Profile!');
					16#0726:
						sMeldSpeich
							:= ('AX5805: PDO-Mapping Achse 1/2: Fehler FSOE COMMAND!');
					16#0727:
						sMeldSpeich
							:= ('AX5805: PDO-Mapping Achse 1: Length_Error!');
					16#0728:
						sMeldSpeich
							:= ('AX5805: PDO-Mapping Achse 1: Fehler STO!');
					16#0729:
						sMeldSpeich
							:= ('AX5805: PDO-Mapping Achse 1: Fehler SS1_1!');
					16#072A:
						sMeldSpeich
							:= ('AX5805: PDO-Mapping Achse 1: Fehler SS2_1!');
					16#072B:
						sMeldSpeich
							:= ('AX5805: PDO-Mapping Achse 1: Fehler SOS_1!');
					16#072C:
						sMeldSpeich
							:= ('AX5805: PDO-Mapping Achse 1: Fehler SSR_1!');
					16#072D:
						sMeldSpeich
							:= ('AX5805: PDO-Mapping Achse 1: Fehler SDIp!');
					16#072E:
						sMeldSpeich
							:= ('AX5805: PDO-Mapping Achse 1: Fehler SDIn!');
					16#072F:
						sMeldSpeich
							:= ('AX5805: PDO-Mapping Achse 1: Fehler Error_ACK!');
					16#0730:
						sMeldSpeich
							:= ('AX5805: PDO-Mapping Achse 1/2: Fehler FSOE CRC0!');
					16#0731:
						sMeldSpeich
							:= ('AX5805: PDO-Mapping Achse 2: Fehler STO!');
					16#0732:
						sMeldSpeich
							:= ('AX5805: PDO-Mapping Achse 2: Fehler SS1_1!');
					16#0733:
						sMeldSpeich
							:= ('AX5805: PDO-Mapping Achse 2: Fehler SS2_1!');
					16#0734:
						sMeldSpeich
							:= ('AX5805: PDO-Mapping Achse 2: Fehler SOS_1!');
					16#0735:
						sMeldSpeich
							:= ('AX5805: PDO-Mapping Achse 2: Fehler SSR_1!');
					16#0736:
						sMeldSpeich
							:= ('AX5805: PDO-Mapping Achse 2: Fehler SDIp!');
					16#0737:
						sMeldSpeich
							:= ('AX5805: PDO-Mapping Achse 2: Fehler SDIn!');
					16#0738:
						sMeldSpeich
							:= ('AX5805: PDO-Mapping Achse 2: Fehler Error_ACK!');
					16#0739:
						sMeldSpeich
							:= ('AX5805: PDO-Mapping Achse 2: Fehler FSOE CRC1!');
					16#073A:
						sMeldSpeich
							:= ('AX5805: PDO-Mapping Achse 1/2: Fehler FSOE ConnID!');
					16#073B:
						sMeldSpeich
							:= ('AX5805: PDO-Mapping Achse 1: Fehler SSM_1_K1!');
					16#073C:
						sMeldSpeich
							:= ('AX5805: PDO-Mapping Achse 2: Fehler SSM_1_K2!');
					16#073D:
						sMeldSpeich
							:= ('AX5805: PDO-Mapping Achse 1: Fehler SSM_2_K1!');
					16#073E:
						sMeldSpeich
							:= ('AX5805: PDO-Mapping Achse 2: Fehler SSM_2_K2!');
					16#0740:
						sMeldSpeich
							:= ('AX5805: Registerkommunikation: Parametrierter Motortyp für Achse1 stimmt nicht mit angeschlossenem Motor überein!');
					16#0741:
						sMeldSpeich
							:= ('AX5805: Registerkommunikation: Parametrierter Motortyp für Achse1 ist unbekannt!');
					16#0742:
						sMeldSpeich
							:= ('AX5805: Registerkommunikation: Parametrierter Motortyp für Achse2 stimmt nicht mit angeschlossenem Motor überein!');
					16#0743:
						sMeldSpeich
							:= ('AX5805: Registerkommunikation: Parametrierter Motortyp für Achse2 ist unbekannt!');
					16#0744:
						sMeldSpeich
							:= ('AX5805: Registerkommunikation: Parametrierte Polpaarzahl für Achse1 stimmt nicht mit angeschlossenem Motor überein!');
					16#0745:
						sMeldSpeich
							:= ('AX5805: Registerkommunikation: Parametrierte Polpaarzahl für Achse2 stimmt nicht mit angeschlossenem Motor überein!');
					16#0746:
						sMeldSpeich
							:= ('AX5805: Registerkommunikation: Parametrierter Motor für Achse1 stimmt nicht mit angeschlossenem Motor überein!');
					16#0747:
						sMeldSpeich
							:= ('AX5805: Registerkommunikation: Parametrierter Motor für Achse2 stimmt nicht mit angeschlossenem Motor überein!');
					16#0748:
						sMeldSpeich
							:= ('AX5805: PDO-Mapping: RXPDO Länge ist falsch!');
					16#0749:
						sMeldSpeich
							:= ('AX5805: PDO-Mapping: TXPDO Länge ist falsch!');
					16#074A:
						sMeldSpeich
							:= ('AX5805: PDO-Mapping: RXPDO Index ist unbekannt!');
					16#074B:
						sMeldSpeich
							:= ('AX5805: PDO-Mapping: TXPDO Index ist unbekannt!');
					16#074C:
						sMeldSpeich
							:= ('AX5805: Die parametrierte Anzahl der Achsen stimmt nicht mit der detektierten überein!');
					16#1001:
						sMeldSpeich
							:= ('AX5805: Eine fehlerhafte Checksumme bei µC1 wurde beim PowerOn Reset ermittelt!');
					16#1002:
						sMeldSpeich
							:= ('AX5805: Eine fehlerhafte Checksumme bei µC2 wurde beim PowerOn Reset ermittelt!');
					16#1003:
						sMeldSpeich
							:= ('AX5805: Eine fehlerhafte Checksumme wurde bei µC1 im laufenden Betrieb ermittelt!');
					16#1004:
						sMeldSpeich
							:= ('AX5805: Eine fehlerhafte Checksumme wurde bei µC2 im laufenden Betrieb ermittelt!');
					16#1011:
						sMeldSpeich
							:= ('AX5805: Fehler beim RAM Test von µC1 ist aufgetreten!');
					16#1012:
						sMeldSpeich
							:= ('AX5805: Fehler beim RAM Test von µC2 ist aufgetreten!');
					16#1013:
						sMeldSpeich
							:= ('AX5805: Fehler beim RAM Test von µC1 ist aufgetreten!');
					16#1014:
						sMeldSpeich
							:= ('AX5805: Fehler beim RAM Test von µC2 ist aufgetreten!');
					16#1021:
						sMeldSpeich
							:= ('AX5805: Der globale Timer arbeitet nicht korrekt!');
					16#1031:
						sMeldSpeich
							:= ('AX5805: Stack-Überläufe werden nicht mehr korrekt abgefangen!');
					16#1032:
						sMeldSpeich
							:= ('AX5805: Stack-Überläufe werden nicht mehr korrekt abgefangen!');
					16#1100:
						sMeldSpeich
							:= ('AX5805: Der Opcode Test von µC1 ist fehlgeschlagen!');
					16#1300:
						sMeldSpeich
							:= ('AX5805: Der Opcode Test von µC2 ist fehlgeschlagen!');
					16#1801:
						sMeldSpeich
							:= ('AX5805: Es wurden unterschiedliche Checksummen bei den TwinSAFE Telegrammen ermittelt!');
					16#1802:
						sMeldSpeich
							:= ('AX5805: Es wurden unterschiedliche Checksummen bei den TwinSAFE Telegrammen ermittelt!');
					16#1803:
						sMeldSpeich
							:= ('AX5805: Es wurde der Defaultcase der Mainschleife von µC1 aufgerufen!');
					16#1804:
						sMeldSpeich
							:= ('AX5805: Es wurde der Defaultcase der Mainschleife von µC2 aufgerufen!');
					16#1805:
						sMeldSpeich
							:= ('AX5805: Die Connection Id ist nicht Null beim Lesen der Projekt CRC!');
					16#1806:
						sMeldSpeich
							:= ('AX5805: Die Connection Id ist nicht Null beim Schreiben der Projekt CRC!');
					16#1807:
						sMeldSpeich
							:= ('AX5805: Es wird auf eine Adresse außerhalb des Herstellbereichs im EEPROM zugegriffen!');
					16#5100:
						sMeldSpeich
							:= ('AX5805: Die Kommunikation zwischen µC1 und µC2 ist gestört!');
					16#5101:
						sMeldSpeich
							:= ('AX5805: High-Prio ISR: Kommunikation unterbrochen: Feedback Schaltnetzteil!');
					16#5102:
						sMeldSpeich
							:= ('AX5805: High-Prio ISR: Kommunikation unterbrochen: Winkel Achse1!');
					16#5103:
						sMeldSpeich
							:= ('AX5805: High-Prio ISR: Kommunikation unterbrochen: Winkel Achse2!');
					16#5104:
						sMeldSpeich
							:= ('AX5805: High-Prio ISR: Kommunikation unterbrochen: zurückgelegter Weg Achse1!');
					16#5105:
						sMeldSpeich
							:= ('AX5805: High-Prio ISR: Kommunikation unterbrochen: zurückgelegter Weg Achse2!');
					16#5106:
						sMeldSpeich
							:= ('AX5805: High-Prio ISR: Kommunikation unterbrochen: Geschwindigkeit Achse1!');
					16#5107:
						sMeldSpeich
							:= ('AX5805: High-Prio ISR: Kommunikation unterbrochen: Geschwindigkeit Achse2!');
					16#5108:
						sMeldSpeich
							:= ('AX5805: High-Prio ISR: Kommunikation unterbrochen: Feedback der Abschaltkanäle!');
					16#5109:
						sMeldSpeich
							:= ('AX5805: Registerkommunikation: AX5000 antwortet nicht rechtzeitig: Controlword!');
					16#510A:
						sMeldSpeich
							:= ('AX5805: Registerkommunikation: AX5000 antwortet nicht rechtzeitig: Statusword!');
					16#510B:
						sMeldSpeich
							:= ('AX5805: Registerkommunikation: AX5000 antwortet nicht rechtzeitig: Registeradresse!');
					16#510C:
						sMeldSpeich
							:= ('AX5805: Registerkommunikation: AX5000 antwortet nicht rechtzeitig: Registerdaten!');
					16#510D:
						sMeldSpeich
							:= ('AX5805: Registerkommunikation: AX5000 antwortet nicht rechtzeitig: CRC!');
					16#510E:
						sMeldSpeich
							:= ('AX5805: Registerkommunikation: Unbekanntes Interface zum AX5000!');
					16#0510F:
						sMeldSpeich
							:= ('AX5805: Registerkommunikation: Das Interface zum AX5000 hat einen Kommunikationsfehler!');
					16#5110 .. 16#5113:
						sMeldSpeich
							:= ('AX5805: Werte konnten nicht ins Register im AX5000 geschrieben werden!');
					16#5114:
						sMeldSpeich
							:= ('AX5805: High-Prio ISR: Externer ADC: es wurde eine unzulässige Adresse gelesen!');
					16#5115:
						sMeldSpeich
							:= ('AX5805: Register-Kommunikation zum AX5000: Telegramm hat einen CRC Fehler!');
					16#5116:
						sMeldSpeich
							:= ('AX5805: High-Prio ISR: Zyklische-Kommunikation zum AX5000: Telegramm hat einen CRC Fehler!');
					16#5117:
						sMeldSpeich
							:= ('AX5805: Registerkommunikation: Adressiertes Register ist unbekannt!');
					16#5118:
						sMeldSpeich
							:= ('AX5805: High-Prio ISR: Zyklische Kommunikation zum AX5000: AX5000 meldet einen Kommunikationsfehler!');
					16#5119:
						sMeldSpeich
							:= ('AX5805: High-Prio ISR: Zyklische-Kommunikation zwischen µC1 und µC2: Kommunikationsfehler!');
					16#5C00:
						sMeldSpeich
							:= ('AX5805: Gemappte Safety Funktionen: Fehler beim Setzen des State!');
					16#5C01:
						sMeldSpeich
							:= ('AX5805: Gemappte Safety Funktionen: Fehler beim Zurücksetzen des State!');
					16#5C02:
						sMeldSpeich
							:= ('AX5805: Gemappte Safety Funktionen: Ungültiges Mapping, Funktion nicht vorhanden!');
					16#5C03:
						sMeldSpeich
							:= ('AX5805: Gemappte Safety Funktionen: Ungültiges Mapping, Instanz nicht vorhanden!');
					16#5E02:
						sMeldSpeich
							:= ('AX5805: Der angeforderte STO-Mode ist ungültig!');
					16#5E03:
						sMeldSpeich
							:= ('AX5805: Fehlerreaktion: Ungültige Fehlerreaktion, Fehlerreaktion nicht vorhanden!');
					16#5E04:
						sMeldSpeich
							:= ('AX5805: Der angeforderte SDI-Mode ist ungültig!');
					16#5F00:
						sMeldSpeich
							:= ('AX5805: Eine fehlerhafte Checksumme wurde beim Vergleich durch µC1 festgestellt!');
					16#5F01:
						sMeldSpeich
							:= ('AX5805: Eine fehlerhafte Checksumme wurde beim Vergleich durch µC2 festgestellt!');
					16#5F02:
						sMeldSpeich
							:= ('AX5805: MC_Test: Timer2 hat Interrupt auf µC1ausgelöst. HighPrioISR wurde nicht rechtzeitig aufgerufen!');
					16#5F03:
						sMeldSpeich
							:= ('AX5805: MC_Test: Timer2 hat Interrupt auf µC2ausgelöst. HighPrioISR wurde nicht rechtzeitig aufgerufen!');
					16#5F04:
						sMeldSpeich
							:= ('AX5805: MC_Test: der Test der Abschaltkanäle ist fehlgeschlagen!');
					16#5F05:
						sMeldSpeich
							:= ('AX5805: Kein SYNC-Signal!');
					16#5F06:
						sMeldSpeich
							:= ('AX5805: Angeforderte Achse nicht bekannt!');
					16#5F07:
						sMeldSpeich
							:= ('AX5805: Der Status des FPGA ist fehlerhaft!');
					16#5F08:
						sMeldSpeich
							:= ('AX5805: Die eingelesenen Winkel von µC1 haben das falsche Format!');
					16#5F09:
						sMeldSpeich
							:= ('AX5805: Die eingelesenen Winkel von µC2 haben das falsche Format!');
					16#5F0A:
						sMeldSpeich
							:= ('AX5805: Unbekannter State angefordert!');
					16#5F0B:
						sMeldSpeich
							:= ('AX5805: Fehler beim Aufstarten!');
					16#5F0C:
						sMeldSpeich
							:= ('AX5805: Fehler bei der Bewegungserkennung!');
					16#6000:
						sMeldSpeich
							:= ('AX5805: Falsche Vendor ID übermittelt!');
					16#6001:
						sMeldSpeich
							:= ('AX5805: Falsche Module ID übermittelt!');
					16#6002:
						sMeldSpeich
							:= ('AX5805: CRC der AX5805 Parameter passt nicht zu der übermittelten CRC (Bitte Parameter kontrollieren und ggf. System Manager Konfiguration aktivieren und Safety Projekt neu in die EL69xx laden).!');
				 END_CASE
				 IF nReadBuf > 0 THEN	(*Erstellen der Fehlermeldung*)
					 arrSafetyKlemmeInfo[nAktKlemme].arrFehler[nFehlerIdx] := TRUE;	
					 arrSafetyKlemmeInfo[nAktKlemme].arrFehlertext[nFehlerIdx] := 	  	
						CONCAT(sMeldSpeich,
						CONCAT(' Achse:',
						CONCAT(INT_TO_STRING(nAktAchse),
						CONCAT('Adresse: ',
							arrSafetyKlemmeInfo[nAktKlemme].sName))));
					 nFehlerIdx := nFehlerIdx + 1;	
				  END_IF
				  bCoeReadError := FALSE;
				 END_IF
			IF nAktAchse < nAnzahlAchsen THEN
				nAktAchse := nAktAchse + 1;
			ELSIF nAktAchse = nAnzahlAchsen THEN
				nAktAchse := 0;
				arrSafetyKlemmeInfo[nAktKlemme].nAnzFehler := nFehlerIdx;
				nFehlerIdx := 0;
				bBusy := FALSE;
				nStateDatenAuslesen := 0;
			END_IF
		END_IF
	END_IF
END_CASE
END_ACTION

ACTION f_AX5806:
CASE nStateDatenAuslesen OF
0:
	(*Auslesen der Anzahl der Achsen*)
	bBusy				:= TRUE;	
	nCoeIndex		:= 16#2F00; (*Anzahl der Achsen*)
	nCoESubIndex	:= 16#1;
	
	fbCoeRead(
	sNetId		:= sEtherCatNetID,
	nSlaveAddr 	:= arrSafetyKlemmeInfo[nAktKlemme].nAdresse,
	nIndex		:= nCoEIndex,
	nSubIndex 	:= nCoESubIndex,
	pDstBuf		:= ADR(nReadBuf),
	cbBufLen		:= SIZEOF(nReadBuf),
	bExecute		:= TRUE,

	bError		=> bCoeReadError,
	nErrId		=> nCoeReadErrId
	);
	
	fbCoeRead(bExecute:= FALSE);
	nAnzahlAchsen := UDINT_TO_INT(nReadBuf);
	
	IF NOT fbCoeRead.bBusy THEN
		nStateDatenAuslesen := nStateDatenAuslesen + 1;
	END_IF
	
1:	
	IF nAktAChse < nAnzahlAchsen THEN
		IF nAktAchse = 0 THEN
			  nAktAchse := 1;
	   END_IF
		
		nCoeIndex		:= 16#FA10; (*Grund der Abschaltung*)
		IF nAktAchse = 1 THEN 
			nCoESubIndex := 16#07;	(*Index Achse 1*)
		ELSE
			nCoeSubIndex := 16#08;	(*Index Achse 2*)
		END_IF
		 
		 fbCoeRead(
		 sNetId		:= sEtherCatNetID,
		 nSlaveAddr := arrSafetyKlemmeInfo[nAktKlemme].nAdresse,
		 nIndex		:= nCoEIndex,
		 nSubIndex 	:= nCoESubIndex,
		 pDstBuf		:= ADR(nReadBuf),
		 cbBufLen		:= SIZEOF(nReadBuf),
		 bExecute		:= TRUE,
	 
		 bError		=> bCoeReadError,
		 nErrId		=> nCoeReadErrId
		 );
			 
		 fbCoeRead(bExecute:= FALSE);
	 
		 IF NOT fbCoeRead.bBusy THEN				(* Baustein ist durchgelaufen *)
			 IF fbCoeRead.bError THEN				(* Wenn ein Error vorliegt, wird dieser ausgegeben; 0 = kein Fehler, 1= Eingang 1; 2= Eingang 2; 3= Eingang 3; 4 = Eingang 4*)
				 nLastErrIDTemp 
					 := fbCoeRead.nErrID;
				 bCoeReadError := TRUE;
			 ELSE
		 (*Fehler-Meldungen - Grund der Abschaltung CoE Objekt 0xFA10:07 und 0xFA10:08*)
		 (*Fehlermeldung aus AX5805.pdf Stand 03.12.2013 - S.101*)
			IF nReadBuf >= 16#100
			 AND nReadBuf < 16#200 THEN
				arrSafetyKlemmeInfo[nAktKlemme].arrFehler[nFehlerIdx] := TRUE;
				arrSafetyKlemmeInfo[nAktKlemme].arrFehlertext[nFehlerIdx] := 
					 CONCAT('AX5805: Das Statuswort wurde falsch berechnet! Achse: ',
					 CONCAT(INT_TO_STRING(nAktAchse),
					 CONCAT('Adresse: ',
						arrSafetyKlemmeInfo[nAktKlemme].sName)));
				nFehlerIdx := nFehlerIdx + 1;
			ELSIF nReadBuf >= 16#200
			 AND nReadBuf < 16#300 THEN
				arrSafetyKlemmeInfo[nAktKlemme].arrFehler[nFehlerIdx] := TRUE;
				arrSafetyKlemmeInfo[nAktKlemme].arrFehlertext[nFehlerIdx] := 
					 CONCAT('AX5805: Die Parameter sind fehlerhaft, wurden noch nicht geladen oder der AX5805 wurde noch nicht zurueckgesetzt (Error_Ack)! Achse: ',
					 CONCAT(INT_TO_STRING(nAktAchse),
					 CONCAT('Adresse: ',
						arrSafetyKlemmeInfo[nAktKlemme].sName)));
				nFehlerIdx := nFehlerIdx + 1;	
			ELSIF nReadBuf >= 16#300
			 AND nReadBuf < 16#400 THEN
				arrSafetyKlemmeInfo[nAktKlemme].arrFehler[nFehlerIdx] := TRUE;
				arrSafetyKlemmeInfo[nAktKlemme].arrFehlertext[nFehlerIdx] := 
					 CONCAT('AX5805: FSOE-Protokoll nicht im State DATA! Achse: ',
					 CONCAT(INT_TO_STRING(nAktAchse),
					 CONCAT('Adresse: ',
						arrSafetyKlemmeInfo[nAktKlemme].sName)));
				nFehlerIdx := nFehlerIdx + 1;
			ELSIF nReadBuf >= 16#400
			 AND nReadBuf < 16#500 THEN
				arrSafetyKlemmeInfo[nAktKlemme].arrFehler[nFehlerIdx] := TRUE;
				arrSafetyKlemmeInfo[nAktKlemme].arrFehlertext[nFehlerIdx] := 
					 CONCAT('AX5805: FSOE-Protokoll nicht im State DATA! Achse: ',
					 CONCAT(INT_TO_STRING(nAktAchse),
					 CONCAT('Adresse: ',
						arrSafetyKlemmeInfo[nAktKlemme].sName)));
				nFehlerIdx := nFehlerIdx + 1;
			 ELSIF nReadBuf >= 16#500
				 AND nReadBuf < 16#600 THEN
					 arrSafetyKlemmeInfo[nAktKlemme].arrFehler[nFehlerIdx] := TRUE;
					 arrSafetyKlemmeInfo[nAktKlemme].arrFehlertext[nFehlerIdx] := 
						  CONCAT('AX5805: FSOE-Protokoll nicht im State DATA! Achse: ',
						  CONCAT(INT_TO_STRING(nAktAchse),
						  CONCAT('Adresse: ',
							 arrSafetyKlemmeInfo[nAktKlemme].sName)));	
					 nFehlerIdx := nFehlerIdx + 1;
			 ELSIF nReadBuf >= 16#600
				 AND nReadBuf < 16#700 THEN
					 arrSafetyKlemmeInfo[nAktKlemme].arrFehler[nFehlerIdx] := TRUE;
					 arrSafetyKlemmeInfo[nAktKlemme].arrFehlertext[nFehlerIdx] := 
						  CONCAT('AX5805: FSOE-Protokoll nicht im State DATA! Achse: ',
						  CONCAT(INT_TO_STRING(nAktAchse),
						  CONCAT('Adresse: ',
							 arrSafetyKlemmeInfo[nAktKlemme].sName)));	
					 nFehlerIdx := nFehlerIdx + 1;
			 ELSIF nReadBuf >= 16#700
				 AND nReadBuf < 16#800 THEN
					 arrSafetyKlemmeInfo[nAktKlemme].arrFehler[nFehlerIdx] := TRUE;
					 arrSafetyKlemmeInfo[nAktKlemme].arrFehlertext[nFehlerIdx] := 
						  CONCAT('AX5805: FSOE-Protokoll nicht im State DATA! Achse: ',
						  CONCAT(INT_TO_STRING(nAktAchse),
						  CONCAT('Adresse: ',
							 arrSafetyKlemmeInfo[nAktKlemme].sName)));	
					 nFehlerIdx := nFehlerIdx + 1;
			 ELSIF nReadBuf >= 16#800
				 AND nReadBuf < 16#900 THEN
					 arrSafetyKlemmeInfo[nAktKlemme].arrFehler[nFehlerIdx] := TRUE;
					 arrSafetyKlemmeInfo[nAktKlemme].arrFehlertext[nFehlerIdx] := 
						  CONCAT('AX5805: FSOE-Protokoll nicht im State DATA! Achse: ',
						  CONCAT(INT_TO_STRING(nAktAchse),
						  CONCAT('Adresse: ',
							 arrSafetyKlemmeInfo[nAktKlemme].sName)));	
					 nFehlerIdx := nFehlerIdx + 1;
			 ELSIF nReadBuf >= 16#5000
				 AND nReadBuf < 16#6800 THEN
					 arrSafetyKlemmeInfo[nAktKlemme].arrFehler[nFehlerIdx] := TRUE;
					 arrSafetyKlemmeInfo[nAktKlemme].arrFehlertext[nFehlerIdx] := 
						  CONCAT('AX5805: FSOE-Protokoll nicht im State DATA! Achse: ',
						  CONCAT(INT_TO_STRING(nAktAchse),
						  CONCAT('Adresse: ',
							 arrSafetyKlemmeInfo[nAktKlemme].sName)));	
					 nFehlerIdx := nFehlerIdx + 1;
			 ELSIF nReadBuf >= 16#6800
				 AND nReadBuf < 16#8000 THEN
					 arrSafetyKlemmeInfo[nAktKlemme].arrFehler[nFehlerIdx] := TRUE;
					 arrSafetyKlemmeInfo[nAktKlemme].arrFehlertext[nFehlerIdx] := 
						  CONCAT('AX5805: FSOE-Protokoll nicht im State DATA! Achse: ',
						  CONCAT(INT_TO_STRING(nAktAchse),
						  CONCAT('Adresse: ',
							 arrSafetyKlemmeInfo[nAktKlemme].sName)));	
					 nFehlerIdx := nFehlerIdx + 1;
			 ELSIF nReadBuf >= 16#8000
				 AND nReadBuf < 16#9000 THEN
					 arrSafetyKlemmeInfo[nAktKlemme].arrFehler[nFehlerIdx] := TRUE;
					 arrSafetyKlemmeInfo[nAktKlemme].arrFehlertext[nFehlerIdx] := 
						  CONCAT('AX5805: FSOE-Protokoll nicht im State DATA! Achse: ',
						  CONCAT(INT_TO_STRING(nAktAchse),
						  CONCAT('Adresse: ',
							 arrSafetyKlemmeInfo[nAktKlemme].sName)));	
					 nFehlerIdx := nFehlerIdx + 1;
			 ELSIF nReadBuf >= 16#9000
				 AND nReadBuf < 16#A000 THEN
					 arrSafetyKlemmeInfo[nAktKlemme].arrFehler[nFehlerIdx] := TRUE;
					 arrSafetyKlemmeInfo[nAktKlemme].arrFehlertext[nFehlerIdx] := 
						  CONCAT('AX5805: FSOE-Protokoll nicht im State DATA! Achse: ',
						  CONCAT(INT_TO_STRING(nAktAchse),
						  CONCAT('Adresse: ',
							 arrSafetyKlemmeInfo[nAktKlemme].sName)));	
					 nFehlerIdx := nFehlerIdx + 1;
			 ELSIF nReadBuf >= 16#A000
				 AND nReadBuf < 16#A800 THEN
					 arrSafetyKlemmeInfo[nAktKlemme].arrFehler[nFehlerIdx] := TRUE;
					 arrSafetyKlemmeInfo[nAktKlemme].arrFehlertext[nFehlerIdx] := 
						  CONCAT('AX5805: FSOE-Protokoll nicht im State DATA! Achse: ',
						  CONCAT(INT_TO_STRING(nAktAchse),
						  CONCAT('Adresse: ',
							 arrSafetyKlemmeInfo[nAktKlemme].sName)));	
					 nFehlerIdx := nFehlerIdx + 1;
			 ELSIF nReadBuf >= 16#A800
				 AND nReadBuf < 16#B800 THEN
					 arrSafetyKlemmeInfo[nAktKlemme].arrFehler[nFehlerIdx] := TRUE;
					 arrSafetyKlemmeInfo[nAktKlemme].arrFehlertext[nFehlerIdx] := 
						  CONCAT('AX5805: FSOE-Protokoll nicht im State DATA! Achse: ',
						  CONCAT(INT_TO_STRING(nAktAchse),
						  CONCAT('Adresse: ',
							 arrSafetyKlemmeInfo[nAktKlemme].sName)));	
					 nFehlerIdx := nFehlerIdx + 1;
			 ELSIF nReadBuf >= 16#B800
				 AND nReadBuf < 16#C800 THEN
					 arrSafetyKlemmeInfo[nAktKlemme].arrFehler[nFehlerIdx] := TRUE;
					 arrSafetyKlemmeInfo[nAktKlemme].arrFehlertext[nFehlerIdx] := 
						  CONCAT('AX5805: FSOE-Protokoll nicht im State DATA! Achse: ',
						  CONCAT(INT_TO_STRING(nAktAchse),
						  CONCAT('Adresse: ',
							 arrSafetyKlemmeInfo[nAktKlemme].sName)));	
					 nFehlerIdx := nFehlerIdx + 1;
			 ELSIF nReadBuf >= 16#C800
				 AND nReadBuf < 16#D000 THEN
					 arrSafetyKlemmeInfo[nAktKlemme].arrFehler[nFehlerIdx] := TRUE;
					 arrSafetyKlemmeInfo[nAktKlemme].arrFehlertext[nFehlerIdx] := 
						  CONCAT('AX5805: FSOE-Protokoll nicht im State DATA! Achse: ',
						  CONCAT(INT_TO_STRING(nAktAchse),
						  CONCAT('Adresse: ',
							 arrSafetyKlemmeInfo[nAktKlemme].sName)));	
					 nFehlerIdx := nFehlerIdx + 1;
			 ELSIF nReadBuf >= 16#D000
				 AND nReadBuf < 16#D100 THEN
					 arrSafetyKlemmeInfo[nAktKlemme].arrFehler[nFehlerIdx] := TRUE;
					 arrSafetyKlemmeInfo[nAktKlemme].arrFehlertext[nFehlerIdx] := 
						  CONCAT('AX5805: FSOE-Protokoll nicht im State DATA! Achse: ',
						  CONCAT(INT_TO_STRING(nAktAchse),
						  CONCAT('Adresse: ',
							 arrSafetyKlemmeInfo[nAktKlemme].sName)));	
					 nFehlerIdx := nFehlerIdx + 1;
			 ELSIF nReadBuf >= 16#D100 THEN
				 arrSafetyKlemmeInfo[nAktKlemme].arrFehler[nFehlerIdx] := TRUE;
				 arrSafetyKlemmeInfo[nAktKlemme].arrFehlertext[nFehlerIdx] := 
					 CONCAT('AX5805: FSOE-Protokoll nicht im State DATA! Achse: ',
					 CONCAT(INT_TO_STRING(nAktAchse),
					 CONCAT('Adresse: ',
						 arrSafetyKlemmeInfo[nAktKlemme].sName)));	
				 nFehlerIdx := nFehlerIdx + 1;
			 END_IF
			 bCoeReadError := FALSE;
			END_IF
			IF nAktAchse < nAnzahlAchsen THEN
				 nAktAchse := nAktAchse + 1;
			ELSIF nAktAchse = nAnzahlAchsen THEN
				 nAktAchse := 0;
				 nStateDatenAuslesen := nStateDatenAuslesen + 1;
			 END_IF
		  END_IF
		END_IF

3:
	IF nAktAchse > nAnzahlAchsen THEN 
   	IF nAktAchse = 0 THEN	(*Index der Achse wird in die Zahl der Achse umgewandelt*)
			  nAktAchse := 1;
	   END_IF
		
	 (*Sensortest-Fehler-Überprüfung*)
		 nCoeIndex		:= 16#FA82; (*Index fuer die Diagnose*)
		 IF nAktAchse = 1 THEN 
			 nCoESubIndex := 16#03;	(*Index Achse 1*)
		 ELSE
			 nCoeSubIndex := 16#04;	(*Index Achse 2*)
		 END_IF
		 (*Auslesen der Diagnose-Informationen*)
		 fbCoeRead(
		 sNetId		:= sEtherCatNetID,
		 nSlaveAddr := arrSafetyKlemmeInfo[nAktKlemme].nAdresse,
		 nIndex		:= nCoEIndex,
		 nSubIndex 	:= nCoESubIndex,
		 pDstBuf		:= ADR(nReadBuf),
		 cbBufLen	:= SIZEOF(nReadBuf),
		 bExecute	:= TRUE,
	 
		 bError		=> bCoeReadError,
		 nErrId		=> nCoeReadErrId
		 );
	 
		 fbCoeRead(bExecute:= FALSE);
		 IF NOT fbCoeRead.bBusy THEN				(* Baustein ist durchgelaufen *)
			 IF fbCoeRead.bError THEN				(* Wenn ein Error vorliegt, wird dieser ausgegeben; 0 = kein Fehler, 1= Eingang 1; 2= Eingang 2; 3= Eingang 3; 4 = Eingang 4*)
				 nLastErrIDTemp 
					 := fbCoeRead.nErrID;
				 bCoeReadError := TRUE;
			 ELSE
				(*Fehler-Meldungen - Grund der Abschaltung CoE Objekt 0xFA82:03 und 0xFA82:04*)
		 		(*Fehlermeldung aus AX5805.pdf Stand 03.12.2013 - S.101*)
				 CASE nReadBuf OF
					16#0000:
						;
					16#0001:
						sMeldSpeich
							:= ('AX5805: Die maximale Temperatur wurde überschritten (µC1)!');
					16#0002:
						sMeldSpeich
							:= ('AX5805: Die maximale Temperatur wurde überschritten (µC2)!');
					16#0003:
						sMeldSpeich
							:= ('AX5805: Die minimale Temperatur wurde unterschritten (µC1)!');
					16#0004:
						sMeldSpeich
							:= ('AX5805: Die minimale Temperatur wurde unterschritten (µC2)!');
					16#0101:
						sMeldSpeich
							:= ('AX5805: Die maximale Versorgungsspannung wurde überschritten (3,3 V)!');
					16#0102:
						sMeldSpeich
							:= ('AX5805: Die maximale Versorgungsspannung wurde überschritten (3,3 V)!');
					16#0103:
						sMeldSpeich
							:= ('AX5805: Die minimale Versorgungsspannung wurde unterschritten (3,3 V)!');
					16#0104:
						sMeldSpeich
							:= ('AX5805: Die minimale Versorgungsspannung wurde unterschritten (3,3 V)!');
					16#0201:
						sMeldSpeich
							:= ('AX5805: Die MCTests von µC1 wurden nicht vollstandig in der vorgegebenen Zeit durchgeführt!');
					16#0202:
						sMeldSpeich
							:= ('AX5805: Die MCTests von µC2 wurden nicht vollstandig in der vorgegebenen Zeit durchgeführt!');
					16#0203:
						sMeldSpeich
							:= ('AX5805: Der globale Timer wurde nicht rechtzeitig aktualisiert!');
					16#0204:
						sMeldSpeich
							:= ('AX5805: Der globale Timer wurde nicht rechtzeitig aktualisiert!');
					16#020C:
						sMeldSpeich
							:= ('AX5805: Das TwinSAFE Modul wurde nicht innerhalb der Watchdogzeit aufgerufen!');
					16#020D:
						sMeldSpeich
							:= ('AX5805: Das TwinSAFE Modul wurde nicht innerhalb der Watchdogzeit aufgerufen!');
					16#020E:
						sMeldSpeich
							:= ('AX5805: Bei µC1 ist ein Reset im Betrieb des Kontrollers aufgetreten µC2 wurde dabei nicht zuruckgesetzt!');
					16#0300:
						sMeldSpeich
							:= ('AX5805: Fehler im SerComP24C2 Modul ist bei der Datenübertragung aufgetreten!');
					16#0401 .. 16#040B:
						sMeldSpeich
							:= ('AX5805: Fehler im SerComP24C1 Modul ist bei der Datenübertragung aufgetreten!');
					16#0501 .. 16#507:
						sMeldSpeich
							:= ('AX5805: Ein Fehler in der Kommunikation mit einem der Temperatursensoren ist aufgetreten!');
					16#0601:
						sMeldSpeich
							:= ('AX5805: Die von µC1 und µC2 ausgegebenen Werte unterscheiden sich!');
					16#0602:
						sMeldSpeich
							:= ('AX5805: Die von µC1 und µC2 ausgegebenen Werte unterscheiden sich!');
					16#0700:
						sMeldSpeich
							:= ('AX5805: Die minimale FPGA Versorgungsspannung wurde unterschritten (5 V)!');
					16#0701:
						sMeldSpeich
							:= ('AX5805: Die maximale FPGA Versorgungsspannung wurde unterschritten (5 V)!');
					16#0710:
						sMeldSpeich
							:= ('AX5805: Bei den Feedback-Kanalen von µC1 wurde ein Fehler detektiert!');
					16#0711:
						sMeldSpeich
							:= ('AX5805: Bei den Feedback-Kanalen von µC2 wurde ein Fehler detektiert!');
					16#0720:
						sMeldSpeich
							:= ('AX5805: Allgemeiner Parameterfehler µC1!');
					16#0721:
						sMeldSpeich
							:= ('AX5805: Allgemeiner Parameterfehler µC2!');
					16#0722:
						sMeldSpeich
							:= ('AX5805: Parameter: Unbekannter Parameterindex µC1 Drive Profile!');
					16#0723:
						sMeldSpeich
							:= ('AX5805: Parameter: Unbekannter Parameterindex µC1 Hersteller spezifisch!');
					16#0724:
						sMeldSpeich
							:= ('AX5805: Parameter: Unbekannter Parameterindex µC2 Drive Profile!');
					16#0725:
						sMeldSpeich
							:= ('AX5805: Parameter: Unbekannter Parameterindex µC2 Drive Profile!');
					16#0726:
						sMeldSpeich
							:= ('AX5805: PDO-Mapping Achse 1/2: Fehler FSOE COMMAND!');
					16#0727:
						sMeldSpeich
							:= ('AX5805: PDO-Mapping Achse 1: Length_Error!');
					16#0728:
						sMeldSpeich
							:= ('AX5805: PDO-Mapping Achse 1: Fehler STO!');
					16#0729:
						sMeldSpeich
							:= ('AX5805: PDO-Mapping Achse 1: Fehler SS1_1!');
					16#072A:
						sMeldSpeich
							:= ('AX5805: PDO-Mapping Achse 1: Fehler SS2_1!');
					16#072B:
						sMeldSpeich
							:= ('AX5805: PDO-Mapping Achse 1: Fehler SOS_1!');
					16#072C:
						sMeldSpeich
							:= ('AX5805: PDO-Mapping Achse 1: Fehler SSR_1!');
					16#072D:
						sMeldSpeich
							:= ('AX5805: PDO-Mapping Achse 1: Fehler SDIp!');
					16#072E:
						sMeldSpeich
							:= ('AX5805: PDO-Mapping Achse 1: Fehler SDIn!');
					16#072F:
						sMeldSpeich
							:= ('AX5805: PDO-Mapping Achse 1: Fehler Error_ACK!');
					16#0730:
						sMeldSpeich
							:= ('AX5805: PDO-Mapping Achse 1/2: Fehler FSOE CRC0!');
					16#0731:
						sMeldSpeich
							:= ('AX5805: PDO-Mapping Achse 2: Fehler STO!');
					16#0732:
						sMeldSpeich
							:= ('AX5805: PDO-Mapping Achse 2: Fehler SS1_1!');
					16#0733:
						sMeldSpeich
							:= ('AX5805: PDO-Mapping Achse 2: Fehler SS2_1!');
					16#0734:
						sMeldSpeich
							:= ('AX5805: PDO-Mapping Achse 2: Fehler SOS_1!');
					16#0735:
						sMeldSpeich
							:= ('AX5805: PDO-Mapping Achse 2: Fehler SSR_1!');
					16#0736:
						sMeldSpeich
							:= ('AX5805: PDO-Mapping Achse 2: Fehler SDIp!');
					16#0737:
						sMeldSpeich
							:= ('AX5805: PDO-Mapping Achse 2: Fehler SDIn!');
					16#0738:
						sMeldSpeich
							:= ('AX5805: PDO-Mapping Achse 2: Fehler Error_ACK!');
					16#0739:
						sMeldSpeich
							:= ('AX5805: PDO-Mapping Achse 2: Fehler FSOE CRC1!');
					16#073A:
						sMeldSpeich
							:= ('AX5805: PDO-Mapping Achse 1/2: Fehler FSOE ConnID!');
					16#073B:
						sMeldSpeich
							:= ('AX5805: PDO-Mapping Achse 1: Fehler SSM_1_K1!');
					16#073C:
						sMeldSpeich
							:= ('AX5805: PDO-Mapping Achse 2: Fehler SSM_1_K2!');
					16#073D:
						sMeldSpeich
							:= ('AX5805: PDO-Mapping Achse 1: Fehler SSM_2_K1!');
					16#073E:
						sMeldSpeich
							:= ('AX5805: PDO-Mapping Achse 2: Fehler SSM_2_K2!');
					16#0740:
						sMeldSpeich
							:= ('AX5805: Registerkommunikation: Parametrierter Motortyp für Achse1 stimmt nicht mit angeschlossenem Motor überein!');
					16#0741:
						sMeldSpeich
							:= ('AX5805: Registerkommunikation: Parametrierter Motortyp für Achse1 ist unbekannt!');
					16#0742:
						sMeldSpeich
							:= ('AX5805: Registerkommunikation: Parametrierter Motortyp für Achse2 stimmt nicht mit angeschlossenem Motor überein!');
					16#0743:
						sMeldSpeich
							:= ('AX5805: Registerkommunikation: Parametrierter Motortyp für Achse2 ist unbekannt!');
					16#0744:
						sMeldSpeich
							:= ('AX5805: Registerkommunikation: Parametrierte Polpaarzahl für Achse1 stimmt nicht mit angeschlossenem Motor überein!');
					16#0745:
						sMeldSpeich
							:= ('AX5805: Registerkommunikation: Parametrierte Polpaarzahl für Achse2 stimmt nicht mit angeschlossenem Motor überein!');
					16#0746:
						sMeldSpeich
							:= ('AX5805: Registerkommunikation: Parametrierter Motor für Achse1 stimmt nicht mit angeschlossenem Motor überein!');
					16#0747:
						sMeldSpeich
							:= ('AX5805: Registerkommunikation: Parametrierter Motor für Achse2 stimmt nicht mit angeschlossenem Motor überein!');
					16#0748:
						sMeldSpeich
							:= ('AX5805: PDO-Mapping: RXPDO Länge ist falsch!');
					16#0749:
						sMeldSpeich
							:= ('AX5805: PDO-Mapping: TXPDO Länge ist falsch!');
					16#074A:
						sMeldSpeich
							:= ('AX5805: PDO-Mapping: RXPDO Index ist unbekannt!');
					16#074B:
						sMeldSpeich
							:= ('AX5805: PDO-Mapping: TXPDO Index ist unbekannt!');
					16#074C:
						sMeldSpeich
							:= ('AX5805: Die parametrierte Anzahl der Achsen stimmt nicht mit der detektierten überein!');
					16#1001:
						sMeldSpeich
							:= ('AX5805: Eine fehlerhafte Checksumme bei µC1 wurde beim PowerOn Reset ermittelt!');
					16#1002:
						sMeldSpeich
							:= ('AX5805: Eine fehlerhafte Checksumme bei µC2 wurde beim PowerOn Reset ermittelt!');
					16#1003:
						sMeldSpeich
							:= ('AX5805: Eine fehlerhafte Checksumme wurde bei µC1 im laufenden Betrieb ermittelt!');
					16#1004:
						sMeldSpeich
							:= ('AX5805: Eine fehlerhafte Checksumme wurde bei µC2 im laufenden Betrieb ermittelt!');
					16#1011:
						sMeldSpeich
							:= ('AX5805: Fehler beim RAM Test von µC1 ist aufgetreten!');
					16#1012:
						sMeldSpeich
							:= ('AX5805: Fehler beim RAM Test von µC2 ist aufgetreten!');
					16#1013:
						sMeldSpeich
							:= ('AX5805: Fehler beim RAM Test von µC1 ist aufgetreten!');
					16#1014:
						sMeldSpeich
							:= ('AX5805: Fehler beim RAM Test von µC2 ist aufgetreten!');
					16#1021:
						sMeldSpeich
							:= ('AX5805: Der globale Timer arbeitet nicht korrekt!');
					16#1031:
						sMeldSpeich
							:= ('AX5805: Stack-Überläufe werden nicht mehr korrekt abgefangen!');
					16#1032:
						sMeldSpeich
							:= ('AX5805: Stack-Überläufe werden nicht mehr korrekt abgefangen!');
					16#1100:
						sMeldSpeich
							:= ('AX5805: Der Opcode Test von µC1 ist fehlgeschlagen!');
					16#1300:
						sMeldSpeich
							:= ('AX5805: Der Opcode Test von µC2 ist fehlgeschlagen!');
					16#1801:
						sMeldSpeich
							:= ('AX5805: Es wurden unterschiedliche Checksummen bei den TwinSAFE Telegrammen ermittelt!');
					16#1802:
						sMeldSpeich
							:= ('AX5805: Es wurden unterschiedliche Checksummen bei den TwinSAFE Telegrammen ermittelt!');
					16#1803:
						sMeldSpeich
							:= ('AX5805: Es wurde der Defaultcase der Mainschleife von µC1 aufgerufen!');
					16#1804:
						sMeldSpeich
							:= ('AX5805: Es wurde der Defaultcase der Mainschleife von µC2 aufgerufen!');
					16#1805:
						sMeldSpeich
							:= ('AX5805: Die Connection Id ist nicht Null beim Lesen der Projekt CRC!');
					16#1806:
						sMeldSpeich
							:= ('AX5805: Die Connection Id ist nicht Null beim Schreiben der Projekt CRC!');
					16#1807:
						sMeldSpeich
							:= ('AX5805: Es wird auf eine Adresse außerhalb des Herstellbereichs im EEPROM zugegriffen!');
					16#5100:
						sMeldSpeich
							:= ('AX5805: Die Kommunikation zwischen µC1 und µC2 ist gestört!');
					16#5101:
						sMeldSpeich
							:= ('AX5805: High-Prio ISR: Kommunikation unterbrochen: Feedback Schaltnetzteil!');
					16#5102:
						sMeldSpeich
							:= ('AX5805: High-Prio ISR: Kommunikation unterbrochen: Winkel Achse1!');
					16#5103:
						sMeldSpeich
							:= ('AX5805: High-Prio ISR: Kommunikation unterbrochen: Winkel Achse2!');
					16#5104:
						sMeldSpeich
							:= ('AX5805: High-Prio ISR: Kommunikation unterbrochen: zurückgelegter Weg Achse1!');
					16#5105:
						sMeldSpeich
							:= ('AX5805: High-Prio ISR: Kommunikation unterbrochen: zurückgelegter Weg Achse2!');
					16#5106:
						sMeldSpeich
							:= ('AX5805: High-Prio ISR: Kommunikation unterbrochen: Geschwindigkeit Achse1!');
					16#5107:
						sMeldSpeich
							:= ('AX5805: High-Prio ISR: Kommunikation unterbrochen: Geschwindigkeit Achse2!');
					16#5108:
						sMeldSpeich
							:= ('AX5805: High-Prio ISR: Kommunikation unterbrochen: Feedback der Abschaltkanäle!');
					16#5109:
						sMeldSpeich
							:= ('AX5805: Registerkommunikation: AX5000 antwortet nicht rechtzeitig: Controlword!');
					16#510A:
						sMeldSpeich
							:= ('AX5805: Registerkommunikation: AX5000 antwortet nicht rechtzeitig: Statusword!');
					16#510B:
						sMeldSpeich
							:= ('AX5805: Registerkommunikation: AX5000 antwortet nicht rechtzeitig: Registeradresse!');
					16#510C:
						sMeldSpeich
							:= ('AX5805: Registerkommunikation: AX5000 antwortet nicht rechtzeitig: Registerdaten!');
					16#510D:
						sMeldSpeich
							:= ('AX5805: Registerkommunikation: AX5000 antwortet nicht rechtzeitig: CRC!');
					16#510E:
						sMeldSpeich
							:= ('AX5805: Registerkommunikation: Unbekanntes Interface zum AX5000!');
					16#0510F:
						sMeldSpeich
							:= ('AX5805: Registerkommunikation: Das Interface zum AX5000 hat einen Kommunikationsfehler!');
					16#5110 .. 16#5113:
						sMeldSpeich
							:= ('AX5805: Werte konnten nicht ins Register im AX5000 geschrieben werden!');
					16#5114:
						sMeldSpeich
							:= ('AX5805: High-Prio ISR: Externer ADC: es wurde eine unzulässige Adresse gelesen!');
					16#5115:
						sMeldSpeich
							:= ('AX5805: Register-Kommunikation zum AX5000: Telegramm hat einen CRC Fehler!');
					16#5116:
						sMeldSpeich
							:= ('AX5805: High-Prio ISR: Zyklische-Kommunikation zum AX5000: Telegramm hat einen CRC Fehler!');
					16#5117:
						sMeldSpeich
							:= ('AX5805: Registerkommunikation: Adressiertes Register ist unbekannt!');
					16#5118:
						sMeldSpeich
							:= ('AX5805: High-Prio ISR: Zyklische Kommunikation zum AX5000: AX5000 meldet einen Kommunikationsfehler!');
					16#5119:
						sMeldSpeich
							:= ('AX5805: High-Prio ISR: Zyklische-Kommunikation zwischen µC1 und µC2: Kommunikationsfehler!');
					16#5C00:
						sMeldSpeich
							:= ('AX5805: Gemappte Safety Funktionen: Fehler beim Setzen des State!');
					16#5C01:
						sMeldSpeich
							:= ('AX5805: Gemappte Safety Funktionen: Fehler beim Zurücksetzen des State!');
					16#5C02:
						sMeldSpeich
							:= ('AX5805: Gemappte Safety Funktionen: Ungültiges Mapping, Funktion nicht vorhanden!');
					16#5C03:
						sMeldSpeich
							:= ('AX5805: Gemappte Safety Funktionen: Ungültiges Mapping, Instanz nicht vorhanden!');
					16#5E02:
						sMeldSpeich
							:= ('AX5805: Der angeforderte STO-Mode ist ungültig!');
					16#5E03:
						sMeldSpeich
							:= ('AX5805: Fehlerreaktion: Ungültige Fehlerreaktion, Fehlerreaktion nicht vorhanden!');
					16#5E04:
						sMeldSpeich
							:= ('AX5805: Der angeforderte SDI-Mode ist ungültig!');
					16#5F00:
						sMeldSpeich
							:= ('AX5805: Eine fehlerhafte Checksumme wurde beim Vergleich durch µC1 festgestellt!');
					16#5F01:
						sMeldSpeich
							:= ('AX5805: Eine fehlerhafte Checksumme wurde beim Vergleich durch µC2 festgestellt!');
					16#5F02:
						sMeldSpeich
							:= ('AX5805: MC_Test: Timer2 hat Interrupt auf µC1ausgelöst. HighPrioISR wurde nicht rechtzeitig aufgerufen!');
					16#5F03:
						sMeldSpeich
							:= ('AX5805: MC_Test: Timer2 hat Interrupt auf µC2ausgelöst. HighPrioISR wurde nicht rechtzeitig aufgerufen!');
					16#5F04:
						sMeldSpeich
							:= ('AX5805: MC_Test: der Test der Abschaltkanäle ist fehlgeschlagen!');
					16#5F05:
						sMeldSpeich
							:= ('AX5805: Kein SYNC-Signal!');
					16#5F06:
						sMeldSpeich
							:= ('AX5805: Angeforderte Achse nicht bekannt!');
					16#5F07:
						sMeldSpeich
							:= ('AX5805: Der Status des FPGA ist fehlerhaft!');
					16#5F08:
						sMeldSpeich
							:= ('AX5805: Die eingelesenen Winkel von µC1 haben das falsche Format!');
					16#5F09:
						sMeldSpeich
							:= ('AX5805: Die eingelesenen Winkel von µC2 haben das falsche Format!');
					16#5F0A:
						sMeldSpeich
							:= ('AX5805: Unbekannter State angefordert!');
					16#5F0B:
						sMeldSpeich
							:= ('AX5805: Fehler beim Aufstarten!');
					16#5F0C:
						sMeldSpeich
							:= ('AX5805: Fehler bei der Bewegungserkennung!');
					16#6000:
						sMeldSpeich
							:= ('AX5805: Falsche Vendor ID übermittelt!');
					16#6001:
						sMeldSpeich
							:= ('AX5805: Falsche Module ID übermittelt!');
					16#6002:
						sMeldSpeich
							:= ('AX5805: CRC der AX5805 Parameter passt nicht zu der übermittelten CRC (Bitte Parameter kontrollieren und ggf. System Manager Konfiguration aktivieren und Safety Projekt neu in die EL69xx laden).!');
				 END_CASE
				 IF nReadBuf > 0 THEN	(*Erstellen der Fehlermeldung*)
					 arrSafetyKlemmeInfo[nAktKlemme].arrFehler[nFehlerIdx] := TRUE;	
					 arrSafetyKlemmeInfo[nAktKlemme].arrFehlertext[nFehlerIdx] := 	  	
						CONCAT(sMeldSpeich,
						CONCAT(' Achse:',
						CONCAT(INT_TO_STRING(nAktAchse),
						CONCAT('Adresse: ',
							arrSafetyKlemmeInfo[nAktKlemme].sName))));
					 nFehlerIdx := nFehlerIdx + 1;	
				  END_IF
				  bCoeReadError := FALSE;
				 END_IF
			IF nAktAchse < nAnzahlAchsen THEN
				nAktAchse := nAktAchse + 1;
			ELSIF nAktAchse = nAnzahlAchsen THEN
				nAktAchse := 0;
				arrSafetyKlemmeInfo[nAktKlemme].nAnzFehler := nFehlerIdx;
				nFehlerIdx := 0;
				bBusy := FALSE;
				nStateDatenAuslesen := 0;
			END_IF
		END_IF
	END_IF
END_CASE
END_ACTION

END_FUNCTION_BLOCK

// POUs/Logging/F_AdsErrorIdToString
// Diese Funktion wandelt einen ADS-Error in ein String um.
FUNCTION F_AdsErrorIdToString : Tc2_System.T_MaxString
VAR_INPUT
	I_nErrorID	: UDINT;
END_VAR

CASE I_nErrorID OF
// Global Error Codes
16#0:	F_AdsErrorIdToString := 'No Error';
16#1:	F_AdsErrorIdToString := 'Internal error';
16#2:	F_AdsErrorIdToString := 'No RTime';
16#3:	F_AdsErrorIdToString := 'Allocation locked memory error';
16#4:	F_AdsErrorIdToString := 'Insert mailbox error';
16#5:	F_AdsErrorIdToString := 'Wrong receive HMSG';
16#6:	F_AdsErrorIdToString := 'target port not found';
16#7:	F_AdsErrorIdToString := 'target machine not found';
16#8:	F_AdsErrorIdToString := 'Unknown command ID';
16#9:	F_AdsErrorIdToString := 'Bad task ID';
16#A:	F_AdsErrorIdToString := 'No IO';
16#B:	F_AdsErrorIdToString := 'Unknown ADS command';
16#C:	F_AdsErrorIdToString := 'Win 32 error';
16#D:	F_AdsErrorIdToString := 'Port not connected';
16#E:	F_AdsErrorIdToString := 'Invalid ADS length';
16#F:	F_AdsErrorIdToString := 'Invalid ADS Net ID';
16#10:	F_AdsErrorIdToString := 'Low Installation level';
16#11:	F_AdsErrorIdToString := 'No debug available';
16#12:	F_AdsErrorIdToString := 'Port disabled';
16#13:	F_AdsErrorIdToString := 'Port already connected';
16#14:	F_AdsErrorIdToString := 'ADS Sync Win32 error';
16#15:	F_AdsErrorIdToString := 'ADS Sync Timeout';
16#16:	F_AdsErrorIdToString := 'ADS Sync AMS error';
16#17:	F_AdsErrorIdToString := 'ADS Sync no index map';
16#18:	F_AdsErrorIdToString := 'Invalid ADS port';
16#19:	F_AdsErrorIdToString := 'No memory';
16#1A:	F_AdsErrorIdToString := 'TCP send error';
16#1B:	F_AdsErrorIdToString := 'Host unreachable';
16#1C:	F_AdsErrorIdToString := 'Invalid AMS fragment';

// Router Error Codes
16#500:	F_AdsErrorIdToString := 'No locked memory can be allocated';
16#501:	F_AdsErrorIdToString := 'The size of the router memory could not be changed';
16#502:	F_AdsErrorIdToString := 'The mailbox has reached the maximum number of possible messages. The current sent message was rejected';
16#503:	F_AdsErrorIdToString := 'The mailbox has reached the maximum number of possible messages. The sent message will not be displayed in the debug monitor';
16#504:	F_AdsErrorIdToString := 'Unknown port type';
16#505:	F_AdsErrorIdToString := 'Router is not initialized';
16#506:	F_AdsErrorIdToString := 'The desired port number is already assigned';
16#507:	F_AdsErrorIdToString := 'Port not registered';
16#508:	F_AdsErrorIdToString := 'The maximum number of Ports reached';
16#509:	F_AdsErrorIdToString := 'Invalid port';
16#50A:	F_AdsErrorIdToString := 'TwinCAT Router not active';

// General ADS Error Codes
16#700: F_AdsErrorIdToString := 'error class <device error>';
16#701: F_AdsErrorIdToString := 'Service is not supported by server';
16#702: F_AdsErrorIdToString := 'invalid index group';
16#703: F_AdsErrorIdToString := 'invalid index offset';
16#704: F_AdsErrorIdToString := 'reading/writing not permitted';
16#705: F_AdsErrorIdToString := 'parameter size not correct';
16#706: F_AdsErrorIdToString := 'invalid parameter value(s)';
16#707: F_AdsErrorIdToString := 'device is not in a ready state';
16#708: F_AdsErrorIdToString := 'device is busy';
16#709: F_AdsErrorIdToString := 'invalid context (must be in Windows)';
16#70A: F_AdsErrorIdToString := 'out of memory';
16#70B: F_AdsErrorIdToString := 'invalid parameter value(s)';
16#70C: F_AdsErrorIdToString := 'not found (files, ...)';
16#70D: F_AdsErrorIdToString := 'syntax error in command or file';
16#70E: F_AdsErrorIdToString := 'objects do not match';
16#70F: F_AdsErrorIdToString := 'object already exists';
16#710: F_AdsErrorIdToString := 'symbol not found';
16#711: F_AdsErrorIdToString := 'symbol version invalid';
16#712: F_AdsErrorIdToString := 'server is in invalid state';
16#713: F_AdsErrorIdToString := 'AdsTransMode not supported';
16#714: F_AdsErrorIdToString := 'Notification handle is invalid';
16#715: F_AdsErrorIdToString := 'Notification client not registered';
16#716: F_AdsErrorIdToString := 'no more notification handles';
16#717: F_AdsErrorIdToString := 'size for watch too big';
16#718: F_AdsErrorIdToString := 'device not initialized';
16#719: F_AdsErrorIdToString := 'device has a timeout';
16#71A: F_AdsErrorIdToString := 'query interface failed';
16#71B: F_AdsErrorIdToString := 'wrong interface required';
16#71C: F_AdsErrorIdToString := 'class ID is invalid';
16#71D: F_AdsErrorIdToString := 'object ID is invalid';
16#71E: F_AdsErrorIdToString := 'request is pending';
16#71F: F_AdsErrorIdToString := 'request is aborted';
16#720: F_AdsErrorIdToString := 'signal warning';
16#721: F_AdsErrorIdToString := 'invalid array index';
16#722: F_AdsErrorIdToString := 'symbol not active';
16#723: F_AdsErrorIdToString := 'access denied';
16#724: F_AdsErrorIdToString := 'missing license';
16#725: F_AdsErrorIdToString := 'license expired';
16#726: F_AdsErrorIdToString := 'license exceeded';
16#727: F_AdsErrorIdToString := 'license invalid';
16#728: F_AdsErrorIdToString := 'license invalid system id';
16#729: F_AdsErrorIdToString := 'license not time limited';
16#72A: F_AdsErrorIdToString := 'license issue time in the future';
16#72B: F_AdsErrorIdToString := 'license time period to long';
16#72C: F_AdsErrorIdToString := 'exception occured during system start';
16#72D: F_AdsErrorIdToString := 'License file read twice';
16#72E: F_AdsErrorIdToString := 'invalid signature';
16#72F: F_AdsErrorIdToString := 'public key certificate';
16#740: F_AdsErrorIdToString := 'Error class <client error>';
16#741: F_AdsErrorIdToString := 'nvalid parameter at service';
16#742: F_AdsErrorIdToString := 'polling list is empty';
16#743: F_AdsErrorIdToString := 'var connection already in use';
16#744: F_AdsErrorIdToString := 'invoke ID in use';
16#745: F_AdsErrorIdToString := 'timeout elapsed';
16#746: F_AdsErrorIdToString := 'error in win32 subsystem';
16#747: F_AdsErrorIdToString := 'Invalid client timeout value';
16#748: F_AdsErrorIdToString := 'ads-port not opened';
16#750: F_AdsErrorIdToString := 'internal error in ads sync';
16#751: F_AdsErrorIdToString := 'hash table overflow';
16#752: F_AdsErrorIdToString := 'key not found in hash';
16#753: F_AdsErrorIdToString := 'no more symbols in cache';
16#754: F_AdsErrorIdToString := 'invalid response received';
16#755: F_AdsErrorIdToString := 'sync port is locked';

//Realtime Error Codes
16#1000:	F_AdsErrorIdToString := 'Internal fatal error in the TwinCAT real-time system';
16#1001:	F_AdsErrorIdToString := 'Timer value not vaild';
16#1002:	F_AdsErrorIdToString := 'Task pointer has the invalid value ZERO';
16#1003:	F_AdsErrorIdToString := 'Task stack pointer has the invalid value ZERO';
16#1004:	F_AdsErrorIdToString := 'The demand task priority is already assigned';
16#1005:	F_AdsErrorIdToString := 'No more free TCB (Task Control Block) available. Maximum number of TCBs is 64';
16#1006:	F_AdsErrorIdToString := 'No more free semaphores available. Maximum number of semaphores is 64';
16#1007:	F_AdsErrorIdToString := 'No more free queue available. Maximum number of queue is 64';
16#100D:	F_AdsErrorIdToString := 'An external synchronization interrupt is already applied';
16#100E:	F_AdsErrorIdToString := 'No external synchronization interrupt applied';
16#100F:	F_AdsErrorIdToString := 'The apply of the external synchronization interrupt failed';
16#1010:	F_AdsErrorIdToString := 'Call of a service function in the wrong context';
16#1017:	F_AdsErrorIdToString := 'Intel VT-x extension is not supported';
16#1018:	F_AdsErrorIdToString := 'Intel VT-x extension is not enabled in system BIOS';
16#1019:	F_AdsErrorIdToString := 'Missing function in Intel VT-x extension';
16#101A:	F_AdsErrorIdToString := 'Enabling Intel VT-x fails';

//TCP Winsock Error Codes
16#274D:	F_AdsErrorIdToString := 'A connection attempt failed because the connected party did not properly respond after a period of time, or established connection failed because connected host has failed to respond.';
16#2751:	F_AdsErrorIdToString := 'No connection could be made because the target machine actively refused it. This error normally occurs when you try to connect to a service which is inactive on a different host - a service without a server application.';
16#274C:	F_AdsErrorIdToString := 'No route to a host. A socket operation was attempted to an unreachable host';
ELSE
	F_AdsErrorIdToString := 'Unbekannter Fehler. Wenn größer Dezimal:10060 möglicherweise Win32 Error Codes';
END_CASE

END_FUNCTION

// POUs/Diverse/F_Skalierung
// Diese Funktion Skaliert einen Eingangswert mit seinen Grenzen, zu einen Ausgangswert mit neuen Grenzen
// Wenn z.B. die neuen Grenzen 0 und 100 sind, dann wird der Eingangswert in Prozent umgerechnet.
FUNCTION F_Skalierung : LREAL
VAR_INPUT
	I_fInput	: LREAL;	// Eingangswert
	I_fMaxIn	: LREAL;	// Obere Grenze vom Eingangswert
	I_fMinIn	: LREAL;	// Untere Grenze vom Eingangswert
	I_fMaxOut: LREAL	:= 100;	// Obere Grenze vom Ausgangswert
	I_fMinOut: LREAL	:= 0;	// Untere Grenze vom Ausgangswert
END_VAR
VAR
END_VAR

IF I_fInput > I_fMaxIn
	OR I_fInput < I_fMinIn
	OR I_fMaxIn = I_fMinIn	// wegen Div0
THEN
	F_Skalierung	:= 0;
	RETURN;
END_IF

F_Skalierung	:= (((I_fInput - I_fMinIn) / (I_fMaxIn - I_fMinIn)) * (I_fMaxOut - I_fMinOut)) + I_fMinOut;

END_FUNCTION

// POUs/Diverse/F_Switchbyte
FUNCTION INTERNAL F_Switchbyte : INT
VAR_INPUT
	nSwitchingBytes:UINT;
END_VAR
VAR
	nHighbyte:WORD;
	nLowByte:WORD;
END_VAR

nHighbyte:= SHR(nSwitchingBytes,8);
nlowbyte:=SHL(nSwitchingBytes,8);
F_Switchbyte:= TO_INT(nhighbyte+nlowbyte);

END_FUNCTION

// POUs/Diverse/FB_Blinker
// Dieser FB erzeugt einen Blinktakt mit gleichlanger on und off Zeit.
FUNCTION_BLOCK FB_Blinker
VAR_INPUT
	I_bStart			: BOOL;	// Blinker aktivieren
	I_tBlinkZeit	: TIME;	// Blinkzeit. Gleichlang an und aus
END_VAR
VAR_OUTPUT
	Q_bOut		: BOOL;	// Ausgang mit blinkverhalten. Erst nach I_tBlinkZeit an.
	tonBlinker1	: Tc2_Standard.TON;	// als Output, damit man die verstrichene Zeit auslesen kann
	tonBlinker2	: Tc2_Standard.TON;	// als Output, damit man die verstrichene Zeit auslesen kann
END_VAR
VAR
END_VAR

tonBlinker1(
	IN	:=
		I_bStart
		AND NOT tonBlinker2.Q,
	PT	:= I_tBlinkZeit,
	Q	=> Q_bOut
);

tonBlinker2(
	IN	:= tonBlinker1.Q,
	PT	:= I_tBlinkZeit
);

END_FUNCTION_BLOCK

// POUs/Diverse/FB_ElectronicFuseIOLink
FUNCTION_BLOCK FB_ElectronicFuseIOLink
VAR_INPUT
	I_arrProcessData			: ARRAY[0..12] OF USINT; 	// Prozessdaten, die die PC-0724-800-0I1 zur Verfügung stellt
	I_sBMK						: STRING;
	
	I_sNETID						: T_AMSNetID;				// AoeNetID des Io-Link-Masters
	I_nIOLinkPort				: UINT;						// Portnummer, an die die Sicherung angeschlossen ist (1,2,3 oder 4)
	I_bErrorQuitt				: BOOL;
END_VAR

VAR_IN_OUT
	IQ_stMeld					: ST_MeldElektrSichg;	
END_VAR

VAR_OUTPUT
	Q_fInputVoltage			: LREAL;					// Eingangsspannung der Sicherung

	Q_arrActCurrent			: ARRAY [1..8] OF LREAL;	// aktueller Strom pro Kanal
	Q_arrSetCurrent			: ARRAY [1..8] OF UINT;		// eingestellter Strom pro Kanal -> wird nur nach SPS-Start ausgelesen
	
	Q_sStatus					: ARRAY [1..8] OF STRING;	// Status der Kanäle
	Q_arrOverCurrent			: ARRAY [1..8] OF BOOL;		// Überstrommeldung
	Q_arrTrippedChannel		: ARRAY [1..8] OF BOOL;		// Auslösemeldung
	
	Q_sGroupMessage			: STRING;					// Sammelmeldung aller Fehlzustände

	Q_bMessageOff						: BOOL;
	Q_bMessageTripped					: BOOL;
	Q_bMessageOver90Percent			: BOOL;
	Q_bMessageOver100Percent		: BOOL;
	Q_bMessageHWFuse					: BOOL;
	Q_bMessageLocalOff				: BOOL;
	Q_bMessageInputVoltageAlarm	: BOOL;
END_VAR

VAR
	arrSetCurrent				: ARRAY [1..8] OF INT;
	arrGetStatus				: ARRAY [1..8] OF USINT;
	nIdx							: INT;
	nInputVoltage				: UINT;
	
	//ADS-Read Set Current
	nIndexCurrent				: WORD;		
	nSubIndexCurrent			: BYTE;		 
	nIdxOffsetCurrent			: UDINT;	
	fbAdsReadCurrent			: AdsRead;
	nReadSetCurrent			: INT;
	nCountCurrent				: INT := 1;
	tonWaitReadCurrent		: TON;
	
	//ADS-Read Status
	nIndexStatus				: WORD;		
	nSubIndexStatus			: BYTE;		 
	nIdxOffsetStatus			: UDINT;	
	fbAdsReadStatus			: AdsRead;
	nReadSetStatus				: INT;
	nCountStatus				: INT := 1;
	rtrigGetStatus				: R_TRIG;
	ftrigGetStatus				: F_TRIG;
	tonWaitGetStatus			: TON;
END_VAR

IF I_sNetID = '0.0.0.0.0.0'
THEN
	RETURN;
ELSE
	a_GetCurrent();
	b_GetStatus();
	z_Output();
	z_Message();
END_IF

ACTION a_GetCurrent:



nIdxOffsetCurrent:=(SHL(WORD_TO_DWORD(nIndexCurrent), 16) OR BYTE_TO_WORD(nSubIndexCurrent)); // merge the to values as shown above

fbAdsReadCurrent(						// Function Block call for adsread
	NETID		:= I_sNetID,
	PORT		:= 4095 + I_nIOLinkPort, // Value in DEC *)(*Port1=>1000Hex=4096DEC ;; Port2=>1001Hex=4097DEC ;; Port3=>1000Hex=Dez4098DEC ;; Port2=>1004Hex=4099DEC 
	IDXGRP	:= 16#F302,				 // Fix value IO-Link Service 
	IDXOFFS 	:= nIdxOffsetCurrent ,			 // Index Subindex 
	LEN		:= SIZEOF(arrSetCurrent[nCountCurrent]),
	DESTADDR	:= ADR(arrSetCurrent[nCountCurrent]),			
	TMOUT		:= 	);
		

CASE nReadSetCurrent OF

0: 	//INIT
	fbAdsReadCurrent.READ	:= FALSE;
	tonWaitReadCurrent(IN := TRUE,
						PT:= T#3S);
	IF tonWaitReadCurrent.Q
	THEN
		tonWaitReadCurrent(IN:= FALSE);
		nReadSetCurrent	:= nReadSetCurrent + 1;
	END_IF

1: // Parameter 1
	nCountCurrent				:= 1;
	nIndexCurrent			:= 16#136;
	fbAdsReadCurrent.READ 	:= TRUE;	
	nReadSetCurrent	:= nReadSetCurrent + 1;
2:
	fbAdsReadCurrent.READ	:=FALSE;
	IF NOT fbAdsReadCurrent.BUSY 
		AND NOT fbAdsReadCurrent.ERR 
	THEN		
		nReadSetCurrent	:= nReadSetCurrent + 1;
	END_IF

3: // Parameter 2
	nCountCurrent				:= 2;
	nIndexCurrent			:= 16#137;
	fbAdsReadCurrent.READ 	:= TRUE;	
	nReadSetCurrent	:= nReadSetCurrent + 1;
4:
	fbAdsReadCurrent.READ	:=FALSE;
	IF NOT fbAdsReadCurrent.BUSY 
		AND NOT fbAdsReadCurrent.ERR 
	THEN		
		nReadSetCurrent	:= nReadSetCurrent + 1;
	END_IF

5: // Parameter 3
	nCountCurrent				:= 3;
	nIndexCurrent			:= 16#138;
	fbAdsReadCurrent.READ 	:= TRUE;	
	nReadSetCurrent	:= nReadSetCurrent + 1;
6:
	fbAdsReadCurrent.READ	:=FALSE;
	IF NOT fbAdsReadCurrent.BUSY 
		AND NOT fbAdsReadCurrent.ERR 
	THEN		
		nReadSetCurrent	:= nReadSetCurrent + 1;
	END_IF

7: // Parameter 4
	nCountCurrent				:= 4;
	nIndexCurrent			:= 16#139;
	fbAdsReadCurrent.READ 	:= TRUE;	
	nReadSetCurrent	:= nReadSetCurrent + 1;
8:
	fbAdsReadCurrent.READ	:=FALSE;
	IF NOT fbAdsReadCurrent.BUSY 
		AND NOT fbAdsReadCurrent.ERR 
	THEN		
		nReadSetCurrent	:= nReadSetCurrent + 1;
	END_IF

9: // Parameter 5
	nCountCurrent				:= 5;
	nIndexCurrent			:= 16#13A;
	fbAdsReadCurrent.READ 	:= TRUE;	
	nReadSetCurrent	:= nReadSetCurrent + 1;
10:
	fbAdsReadCurrent.READ	:=FALSE;
	IF NOT fbAdsReadCurrent.BUSY 
		AND NOT fbAdsReadCurrent.ERR 
	THEN		
		nReadSetCurrent	:= nReadSetCurrent + 1;
	END_IF

11: // Parameter 6
	nCountCurrent				:= 6;
	nIndexCurrent			:= 16#13B;
	fbAdsReadCurrent.READ 	:= TRUE;	
	nReadSetCurrent	:= nReadSetCurrent + 1;
12:
	fbAdsReadCurrent.READ	:=FALSE;
	IF NOT fbAdsReadCurrent.BUSY 
		AND NOT fbAdsReadCurrent.ERR 
	THEN		
		nReadSetCurrent	:= nReadSetCurrent + 1;
	END_IF

13: // Parameter 7
	nCountCurrent				:= 7;
	nIndexCurrent			:= 16#13C;
	fbAdsReadCurrent.READ 	:= TRUE;	
	nReadSetCurrent	:= nReadSetCurrent + 1;
14:
	fbAdsReadCurrent.READ	:=FALSE;
	IF NOT fbAdsReadCurrent.BUSY 
		AND NOT fbAdsReadCurrent.ERR 
	THEN		
		nReadSetCurrent	:= nReadSetCurrent + 1;
	END_IF

15: // Parameter 8
	nCountCurrent				:= 8;
	nIndexCurrent			:= 16#13D;
	fbAdsReadCurrent.READ 	:= TRUE;	
	nReadSetCurrent	:= nReadSetCurrent + 1;
16:
	fbAdsReadCurrent.READ	:=FALSE;
	IF NOT fbAdsReadCurrent.BUSY 
		AND NOT fbAdsReadCurrent.ERR 
	THEN		
		nReadSetCurrent	:= nReadSetCurrent + 1;
	END_IF
END_CASE

Q_arrSetCurrent[1]	:= TO_UINT(F_Switchbyte(INT_TO_UINT(arrSetCurrent[1])));
Q_arrSetCurrent[2]	:= TO_UINT(F_Switchbyte(INT_TO_UINT(arrSetCurrent[2])));
Q_arrSetCurrent[3]	:= TO_UINT(F_Switchbyte(INT_TO_UINT(arrSetCurrent[3])));
Q_arrSetCurrent[4]	:= TO_UINT(F_Switchbyte(INT_TO_UINT(arrSetCurrent[4])));
Q_arrSetCurrent[5]	:= TO_UINT(F_Switchbyte(INT_TO_UINT(arrSetCurrent[5])));
Q_arrSetCurrent[6]	:= TO_UINT(F_Switchbyte(INT_TO_UINT(arrSetCurrent[6])));
Q_arrSetCurrent[7]	:= TO_UINT(F_Switchbyte(INT_TO_UINT(arrSetCurrent[7])));
Q_arrSetCurrent[8]	:= TO_UINT(F_Switchbyte(INT_TO_UINT(arrSetCurrent[8])));
END_ACTION

ACTION b_GetStatus:


nIdxOffsetStatus:=(SHL(WORD_TO_DWORD(nIndexStatus), 16) OR BYTE_TO_WORD(nSubIndexStatus)); // merge the to values as shown above

fbAdsReadStatus(						// Function Block call for adsread
	NETID		:= I_sNetID,
	PORT		:= 4095 + I_nIOLinkPort, // Value in DEC *)(*Port1=>1000Hex=4096DEC ;; Port2=>1001Hex=4097DEC ;; Port3=>1000Hex=Dez4098DEC ;; Port2=>1004Hex=4099DEC 
	IDXGRP		:= 16#F302,				 // Fix value IO-Link Service 
	IDXOFFS 	:= nIdxOffsetStatus ,			 // Index Subindex 
	LEN			:= SIZEOF(arrGetStatus[nCountStatus]),
	DESTADDR	:= ADR(arrGetStatus[nCountStatus]),			
	TMOUT		:= 	);
	
rtrigGetStatus(CLK:= Q_bMessageOff);
ftrigGetStatus(CLK:= Q_bMessageOff);

IF rtrigGetStatus.Q
	OR ftrigGetStatus.Q
THEN
	nReadSetStatus	:= 0;
END_IF
	

CASE nReadSetStatus OF

0: 	//INIT
	fbAdsReadStatus.READ	:= FALSE;
	tonWaitGetStatus(IN:= TRUE,
			PT:= T#500MS);
	IF tonWaitGetStatus.Q
	THEN
		tonWaitGetStatus(IN:= FALSE);
		nReadSetStatus	:= nReadSetStatus + 1;
	END_IF

1: // Parameter 1
	nCountStatus			:= 1;
	nIndexStatus			:= 16#259;
	fbAdsReadStatus.READ 	:= TRUE;	
	nReadSetStatus	:= nReadSetStatus + 1;
2:
	fbAdsReadStatus.READ	:=FALSE;
	IF NOT fbAdsReadStatus.BUSY 
		AND NOT fbAdsReadStatus.ERR 
	THEN		
		nReadSetStatus	:= nReadSetStatus + 1;
	END_IF

3: // Parameter 2
	nCountStatus				:= 2;
	nIndexStatus			:= 16#25A;
	fbAdsReadStatus.READ 	:= TRUE;	
	nReadSetStatus	:= nReadSetStatus + 1;
4:
	fbAdsReadStatus.READ	:=FALSE;
	IF NOT fbAdsReadStatus.BUSY 
		AND NOT fbAdsReadStatus.ERR 
	THEN		
		nReadSetStatus	:= nReadSetStatus + 1;
	END_IF

5: // Parameter 3
	nCountStatus				:= 3;
	nIndexStatus			:= 16#25B;
	fbAdsReadStatus.READ 	:= TRUE;	
	nReadSetStatus	:= nReadSetStatus + 1;
6:
	fbAdsReadStatus.READ	:=FALSE;
	IF NOT fbAdsReadStatus.BUSY 
		AND NOT fbAdsReadStatus.ERR 
	THEN		
		nReadSetStatus	:= nReadSetStatus + 1;
	END_IF

7: // Parameter 4
	nCountStatus				:= 4;
	nIndexStatus			:= 16#25C;
	fbAdsReadStatus.READ 	:= TRUE;	
	nReadSetStatus	:= nReadSetStatus + 1;
8:
	fbAdsReadStatus.READ	:=FALSE;
	IF NOT fbAdsReadStatus.BUSY 
		AND NOT fbAdsReadStatus.ERR 
	THEN		
		nReadSetStatus	:= nReadSetStatus + 1;
	END_IF

9: // Parameter 5
	nCountStatus				:= 5;
	nIndexStatus			:= 16#25D;
	fbAdsReadStatus.READ 	:= TRUE;	
	nReadSetStatus	:= nReadSetStatus + 1;
10:
	fbAdsReadStatus.READ	:=FALSE;
	IF NOT fbAdsReadStatus.BUSY 
		AND NOT fbAdsReadStatus.ERR 
	THEN		
		nReadSetStatus	:= nReadSetStatus + 1;
	END_IF

11: // Parameter 6
	nCountStatus				:= 6;
	nIndexStatus			:= 16#25E;
	fbAdsReadStatus.READ 	:= TRUE;	
	nReadSetStatus	:= nReadSetStatus + 1;
12:
	fbAdsReadStatus.READ	:=FALSE;
	IF NOT fbAdsReadStatus.BUSY 
		AND NOT fbAdsReadStatus.ERR 
	THEN		
		nReadSetStatus	:= nReadSetStatus + 1;
	END_IF

13: // Parameter 7
	nCountStatus				:= 7;
	nIndexStatus			:= 16#25F;
	fbAdsReadStatus.READ 	:= TRUE;	
	nReadSetStatus	:= nReadSetStatus + 1;
14:
	fbAdsReadStatus.READ	:=FALSE;
	IF NOT fbAdsReadStatus.BUSY 
		AND NOT fbAdsReadStatus.ERR 
	THEN		
		nReadSetStatus	:= nReadSetStatus + 1;
	END_IF

15: // Parameter 8
	nCountStatus				:= 8;
	nIndexStatus			:= 16#260;
	fbAdsReadStatus.READ 	:= TRUE;	
	nReadSetStatus	:= nReadSetStatus + 1;
16:
	fbAdsReadStatus.READ	:=FALSE;
	IF NOT fbAdsReadStatus.BUSY 
		AND NOT fbAdsReadStatus.ERR 
	THEN		
		nReadSetStatus	:= 999;
	END_IF
END_CASE

FOR nIdx := 1 TO 8 DO
	CASE arrGetStatus[nIdx] OF
		0:	Q_sStatus[nIdx] := 'Nicht verbunden';
		1:	Q_sStatus[nIdx] := 'Ausgeschaltet über Schnittstelle';
		2:	Q_sStatus[nIdx] := 'Eingeschaltet';
		3:	Q_sStatus[nIdx] := 'Ausgelöst';
		6:	Q_sStatus[nIdx] := 'Strom > 90% Nenn';
		14:	Q_sStatus[nIdx] := 'Strom > 100% Nenn';
		18:	Q_sStatus[nIdx] := 'Hardware Fehler';
		20:	Q_sStatus[nIdx] := 'Thermische Entspannung';
		50:	Q_sStatus[nIdx] := 'Ausgeschaltet über Taster';
		
	END_CASE	

END_FOR
END_ACTION

ACTION z_Message:
Q_sGroupMessage	:= '';

IF Q_bMessageHWFuse
THEN
	Q_sGroupMessage		:= CONCAT(Q_sGroupMessage,'| Hardwarefehler!');
END_IF

IF Q_bMessageInputVoltageAlarm
THEN
	Q_sGroupMessage		:=  CONCAT(Q_sGroupMessage,'| Eingangsspannung ist mit ');
	Q_sGroupMessage		:=  CONCAT(Q_sGroupMessage, LREAL_TO_STRING(Q_fInputVoltage));
	Q_sGroupMessage		:=  CONCAT(Q_sGroupMessage, ' V zu gering');
END_IF
IF Q_bMessageLocalOff
	AND nReadSetStatus = 999
THEN	
	FOR nIdx:= 1 TO 8 DO
		IF arrGetStatus[nIdx] = 50
		THEN
			EXIT;
		END_IF
	END_FOR
	Q_sGroupMessage		:= CONCAT(Q_sGroupMessage,'| Channel '); 
	Q_sGroupMessage		:= CONCAT(Q_sGroupMessage, INT_TO_STRING(nIdx));
	Q_sGroupMessage		:= CONCAT(Q_sGroupMessage,' über Taster ausgeschaltet!');	
END_IF

FOR nIdx:= 1 TO 8 DO
	IF Q_arrTrippedChannel[nIdx]
	THEN
		Q_sGroupMessage		:= CONCAT(Q_sGroupMessage,'| Channel '); 
		Q_sGroupMessage		:= CONCAT(Q_sGroupMessage, INT_TO_STRING(nIdx));
		Q_sGroupMessage		:= CONCAT(Q_sGroupMessage,' hat ausgelößt!');	
	END_IF
	IF Q_arrOverCurrent[nIdx]
	THEN
		Q_sGroupMessage		:= CONCAT(Q_sGroupMessage,'| Channel '); 
		Q_sGroupMessage		:= CONCAT(Q_sGroupMessage, INT_TO_STRING(nIdx));
		Q_sGroupMessage		:= CONCAT(Q_sGroupMessage,' meldet Überstrom!');	
		Q_sGroupMessage		:= CONCAT(Q_sGroupMessage,' Eingestellter Wert: ');	
		Q_sGroupMessage		:= CONCAT(Q_sGroupMessage ,LREAL_TO_STRING(Q_arrSetCurrent [nIdx]/1000));	
		Q_sGroupMessage		:= CONCAT(Q_sGroupMessage ,' A < Istwert ');	
		Q_sGroupMessage		:= CONCAT(Q_sGroupMessage ,LREAL_TO_STRING(Q_arrActCurrent [nIdx]));	
		Q_sGroupMessage		:= CONCAT(Q_sGroupMessage ,' A!');	
	END_IF
END_FOR
END_ACTION

ACTION z_Output:
nInputVoltage	:= SHL((TO_UINT(I_arrProcessData[1])),8) +I_arrProcessData[2];
Q_fInputVoltage	:= UINT_TO_LREAL(nInputVoltage)/100;

FOR nIdx := 1 TO 8 DO
	Q_arrActCurrent[nIdx]	:= USINT_TO_LREAL(I_arrProcessData[nIdx+2])/10;
END_FOR
IF I_arrProcessData[11].0
THEN
	Q_arrOverCurrent[1] := TRUE;
END_IF
IF I_arrProcessData[11].1
THEN
	Q_arrOverCurrent[2] := TRUE;
END_IF
IF I_arrProcessData[11].2
THEN
	Q_arrOverCurrent[3] := TRUE;
END_IF
IF I_arrProcessData[11].3
THEN
	Q_arrOverCurrent[4] := TRUE;
END_IF
IF I_arrProcessData[11].4
THEN
	Q_arrOverCurrent[5] := TRUE;
END_IF
IF I_arrProcessData[11].5
THEN
	Q_arrOverCurrent[6] := TRUE;
END_IF
IF I_arrProcessData[11].6
THEN
	Q_arrOverCurrent[7] := TRUE;
END_IF
IF I_arrProcessData[11].7
THEN
	Q_arrOverCurrent[8] := TRUE;
END_IF


IF I_arrProcessData[12].0
THEN
	Q_arrTrippedChannel[1] := TRUE;
END_IF
IF I_arrProcessData[12].1
THEN
	Q_arrTrippedChannel[2] := TRUE;
END_IF
IF I_arrProcessData[12].2
THEN
	Q_arrTrippedChannel[3] := TRUE;
END_IF
IF I_arrProcessData[12].3
THEN
	Q_arrTrippedChannel[4] := TRUE;
END_IF
IF I_arrProcessData[12].4
THEN
	Q_arrTrippedChannel[5] := TRUE;
END_IF
IF I_arrProcessData[12].5
THEN
	Q_arrTrippedChannel[6] := TRUE;
END_IF
IF I_arrProcessData[12].6
THEN
	Q_arrTrippedChannel[7] := TRUE;
END_IF
IF I_arrProcessData[12].7
THEN
	Q_arrTrippedChannel[8] := TRUE;
END_IF


IF I_bErrorQuitt
THEN
	FOR nIdx:= 1 TO 8 DO	
		Q_arrOverCurrent[nIdx] 		:= FALSE;
		Q_arrTrippedChannel[nIdx] 	:= FALSE;
	END_FOR
END_IF

Q_bMessageOff					:= I_arrProcessData[0].0;
Q_bMessageTripped				:= I_arrProcessData[0].1;
Q_bMessageOver90Percent			:= I_arrProcessData[0].2;
Q_bMessageOver100Percent		:= I_arrProcessData[0].3;
Q_bMessageHWFuse				:= I_arrProcessData[0].4;
Q_bMessageLocalOff				:= I_arrProcessData[0].5;
Q_bMessageInputVoltageAlarm		:= I_arrProcessData[0].6;

IQ_stMeld.SourceName	:= 'Schaltschrank';
IQ_stMeld.sBMK			:= I_sBMK;
IQ_stMeld.bMeldAusg	:= Q_sGroupMessage <> '';
IQ_stMeld.sText		:= Q_sGroupMessage;
END_ACTION

END_FUNCTION_BLOCK

